LIN {X 0,Y 235.007,Z 550.304,A -85,B 0,C 180,E1 -20010.011,E2 -20010.011} C_VEL
LIN {X 0,Y 236.518,Z 558.697,A -85,B 0,C 180,E1 -20011.333,E2 -20011.333} C_VEL
LIN {X 0,Y 237.232,Z 567.162,A -85,B 0,C 180,E1 -20012.793,E2 -20012.793} C_VEL
LIN {X 0,Y 237.343,Z 573.309,A -85,B 0,C 180,E1 -20013.991,E2 -20013.991} C_VEL
LIN {X 0,Y 235.455,Z 581.31,A -85,B 0,C 180,E1 -20015.572,E2 -20015.572} C_VEL
LIN {X 0,Y 233.143,Z 590.008,A -85,B 0,C 180,E1 -20017.763,E2 -20017.763} C_VEL
LIN {X 0,Y 231.134,Z 596.788,A -85,B 0,C 180,E1 -20020.021,E2 -20020.021} C_VEL
LIN {X 0,Y 230.008,Z 600.386,A -85,B 0,C 180,E1 -20021.472,E2 -20021.472} C_VEL
LIN {X 0,Y 228.59,Z 604.847,A -85,B 0,C 180,E1 -20023.737,E2 -20023.737} C_VEL
LIN {X 0,Y 227.388,Z 608.392,A -85,B 0,C 180,E1 -20026.131,E2 -20026.131} C_VEL
LIN {X 0,Y 226.673,Z 610.489,A -85,B 0,C 180,E1 -20028.084,E2 -20028.084} C_VEL
LIN {X 0,Y 226.284,Z 611.528,A -85,B 0,C 180,E1 -20029.289,E2 -20029.289} C_VEL
LIN {X 0,Y 225.779,Z 612.678,A -85,B 0,C 180,E1 -20031.496,E2 -20031.496} C_VEL
LIN {X 0,Y 225.391,Z 613.018,A -85,B 0,C 180,E1 -20034.166,E2 -20034.166} C_VEL
LIN {X 0,Y 225.298,Z 612.689,A -85,B 0,C 180,E1 -20035.84,E2 -20035.84} C_VEL
LIN {X 0,Y 225.374,Z 611.591,A -85,B 0,C 180,E1 -20037.985,E2 -20037.985} C_VEL
LIN {X 0,Y 225.744,Z 609.19,A -85,B 0,C 180,E1 -20040.659,E2 -20040.659} C_VEL
LIN {X 0,Y 226.275,Z 605.609,A -85,B 0,C 180,E1 -20043.233,E2 -20043.233} C_VEL
LIN {X 0,Y 226.922,Z 600.806,A -85,B 0,C 180,E1 -20045.771,E2 -20045.771} C_VEL
LIN {X 0,Y 227.707,Z 595.856,A -85,B 0,C 180,E1 -20047.809,E2 -20047.809} C_VEL
LIN {X 0,Y 228.959,Z 588.315,A -85,B 0,C 180,E1 -20050.265,E2 -20050.265} C_VEL
LIN {X 0,Y 230.164,Z 580.492,A -85,B 0,C 180,E1 -20052.22,E2 -20052.22} C_VEL
LIN {X 0,Y 231.31,Z 573.319,A -85,B 0,C 180,E1 -20053.676,E2 -20053.676} C_VEL
LIN {X 0,Y 232.129,Z 566.346,A -85,B 0,C 180,E1 -20054.862,E2 -20054.862} C_VEL
LIN {X 0,Y 231.344,Z 557.78,A -85,B 0,C 180,E1 -20056.158,E2 -20056.158} C_VEL
LIN {X 0,Y 230.265,Z 549.339,A -85,B 0,C 180,E1 -20057.215,E2 -20057.215} C_VEL
LIN {X 0,Y 228.715,Z 539.614,A -85,B 0,C 180,E1 -20058.197,E2 -20058.197} C_VEL
LIN {X 0,Y 227.156,Z 531.405,A -85,B 0,C 180,E1 -20058.85,E2 -20058.85} C_VEL
LIN {X 0,Y 227.603,Z 525.746,A -85,B 0,C 180,E1 -20062.904,E2 -20062.904} C_VEL
LIN {X 0,Y 227.945,Z 520.793,A -85,B 0,C 180,E1 -20066.464,E2 -20066.464} C_VEL
LIN {X 0,Y 228.369,Z 516.852,A -85,B 0,C 180,E1 -20069.338,E2 -20069.338} C_VEL
LIN {X 0,Y 228.557,Z 516.827,A -85,B 0,C 180,E1 -20071.761,E2 -20071.761} C_VEL
LIN {X 0,Y 228.36,Z 516.851,A -85,B 0,C 180,E1 -20077.07,E2 -20077.07} C_VEL
LIN {X 0,Y 228.173,Z 516.875,A -85,B 0,C 180,E1 -20080.649,E2 -20080.649} C_VEL
LIN {X 0,Y 228.059,Z 516.89,A -85,B 0,C 180,E1 -20086.101,E2 -20086.101} C_VEL
LIN {X 0,Y 227.943,Z 516.901,A -85,B 0,C 180,E1 -20089.824,E2 -20089.824} C_VEL
LIN {X 0,Y 227.914,Z 516.904,A -85,B 0,C 180,E1 -20093.632,E2 -20093.632} C_VEL
LIN {X 0,Y 227.887,Z 516.909,A -85,B 0,C 180,E1 -20097.554,E2 -20097.554} C_VEL
LIN {X 0,Y 227.873,Z 516.912,A -85,B 0,C 180,E1 -20101.621,E2 -20101.621} C_VEL
LIN {X 0,Y 227.899,Z 516.907,A -85,B 0,C 180,E1 -20105.867,E2 -20105.867} C_VEL
LIN {X 0,Y 227.866,Z 516.912,A -85,B 0,C 180,E1 -20110.367,E2 -20110.367} C_VEL
LIN {X 0,Y 227.899,Z 516.903,A -85,B 0,C 180,E1 -20112.721,E2 -20112.721} C_VEL
LIN {X 0,Y 227.908,Z 516.908,A -85,B 0,C 180,E1 -20117.737,E2 -20117.737} C_VEL
LIN {X 0,Y 227.87,Z 516.91,A -85,B 0,C 180,E1 -20121.914,E2 -20121.914} C_VEL
LIN {X 0,Y 227.889,Z 516.909,A -85,B 0,C 180,E1 -20126.372,E2 -20126.372} C_VEL
LIN {X 0,Y 227.902,Z 516.907,A -85,B 0,C 180,E1 -20130.435,E2 -20130.435} C_VEL
LIN {X 0,Y 227.926,Z 516.904,A -85,B 0,C 180,E1 -20134.425,E2 -20134.425} C_VEL
LIN {X 0,Y 227.96,Z 516.901,A -85,B 0,C 180,E1 -20138.287,E2 -20138.287} C_VEL
LIN {X 0,Y 228.032,Z 516.89,A -85,B 0,C 180,E1 -20142.825,E2 -20142.825} C_VEL
LIN {X 0,Y 228.092,Z 516.885,A -85,B 0,C 180,E1 -20147.544,E2 -20147.544} C_VEL
LIN {X 0,Y 228.323,Z 516.854,A -85,B 0,C 180,E1 -20151.147,E2 -20151.147} C_VEL
LIN {X 0,Y 228.356,Z 516.85,A -85,B 0,C 180,E1 -20152.928,E2 -20152.928} C_VEL
LIN {X 0,Y 228.553,Z 516.82,A -85,B 0,C 180,E1 -20158.238,E2 -20158.238} C_VEL
LIN {X 0,Y 228.553,Z 516.827,A -85,B 0,C 180,E1 -20161.762,E2 -20161.762} C_VEL
LIN {X 0,Y 228.356,Z 516.85,A -85,B 0,C 180,E1 -20167.071,E2 -20167.071} C_VEL
LIN {X 0,Y 228.169,Z 516.874,A -85,B 0,C 180,E1 -20170.65,E2 -20170.65} C_VEL
LIN {X 0,Y 228.055,Z 516.889,A -85,B 0,C 180,E1 -20176.102,E2 -20176.102} C_VEL
LIN {X 0,Y 227.94,Z 516.906,A -85,B 0,C 180,E1 -20179.825,E2 -20179.825} C_VEL
LIN {X 0,Y 227.912,Z 516.911,A -85,B 0,C 180,E1 -20183.633,E2 -20183.633} C_VEL
LIN {X 0,Y 227.883,Z 516.914,A -85,B 0,C 180,E1 -20187.555,E2 -20187.555} C_VEL
LIN {X 0,Y 227.87,Z 516.915,A -85,B 0,C 180,E1 -20191.622,E2 -20191.622} C_VEL
LIN {X 0,Y 227.898,Z 516.909,A -85,B 0,C 180,E1 -20195.869,E2 -20195.869} C_VEL
LIN {X 0,Y 227.835,Z 516.916,A -85,B 0,C 180,E1 -20200.374,E2 -20200.374} C_VEL
LIN {X 0,Y 227.846,Z 516.915,A -85,B 0,C 180,E1 -20204.812,E2 -20204.812} C_VEL
LIN {X 0,Y 227.905,Z 516.909,A -85,B 0,C 180,E1 -20207.74,E2 -20207.74} C_VEL
LIN {X 0,Y 228.276,Z 516.988,A -85,B 0,C 180,E1 -20213.175,E2 -20213.175} C_VEL
LIN {X 0,Y 228.987,Z 520.827,A -85,B 0,C 180,E1 -20216.466,E2 -20216.466} C_VEL
LIN {X 0,Y 228.999,Z 523.333,A -85,B 0,C 180,E1 -20218.553,E2 -20218.553} C_VEL
LIN {X 0,Y 228.777,Z 524.324,A -85,B 0,C 180,E1 -20219.365,E2 -20219.365} C_VEL
LIN {X 0,Y 227.83,Z 525.477,A -85,B 0,C 180,E1 -20220.287,E2 -20220.287} C_VEL
LIN {X 0,Y 224.604,Z 527.281,A -85,B 0,C 180,E1 -20221.709,E2 -20221.709} C_VEL
LIN {X 0,Y 221.378,Z 529.082,A -85,B 0,C 180,E1 -20223.169,E2 -20223.169} C_VEL
LIN {X 0,Y 220.469,Z 530.23,A -85,B 0,C 180,E1 -20224.136,E2 -20224.136} C_VEL
LIN {X 0,Y 220.27,Z 531.464,A -85,B 0,C 180,E1 -20225.118,E2 -20225.118} C_VEL
LIN {X 0,Y 220.333,Z 537.076,A -85,B 0,C 180,E1 -20226.608,E2 -20226.608} C_VEL
LIN {X 0,Y 222.079,Z 549.396,A -85,B 0,C 180,E1 -20227.381,E2 -20227.381} C_VEL
LIN {X 0,Y 223.02,Z 560.406,A -85,B 0,C 180,E1 -20228.39,E2 -20228.39} C_VEL
LIN {X 0,Y 223.44,Z 568.042,A -85,B 0,C 180,E1 -20229.278,E2 -20229.278} C_VEL
LIN {X 0,Y 223.685,Z 576.512,A -85,B 0,C 180,E1 -20230.488,E2 -20230.488} C_VEL
LIN {X 0,Y 223.645,Z 584.746,A -85,B 0,C 180,E1 -20231.923,E2 -20231.923} C_VEL
LIN {X 0,Y 222.623,Z 592.352,A -85,B 0,C 180,E1 -20233.495,E2 -20233.495} C_VEL
LIN {X 0,Y 221.149,Z 601.055,A -85,B 0,C 180,E1 -20235.743,E2 -20235.743} C_VEL
LIN {X 0,Y 220.121,Z 607.776,A -85,B 0,C 180,E1 -20238.023,E2 -20238.023} C_VEL
LIN {X 0,Y 219.513,Z 612.188,A -85,B 0,C 180,E1 -20239.859,E2 -20239.859} C_VEL
LIN {X 0,Y 218.864,Z 617.345,A -85,B 0,C 180,E1 -20242.621,E2 -20242.621} C_VEL
LIN {X 0,Y 218.62,Z 620.919,A -85,B 0,C 180,E1 -20245.244,E2 -20245.244} C_VEL
LIN {X 0,Y 218.634,Z 623.486,A -85,B 0,C 180,E1 -20248.159,E2 -20248.159} C_VEL
LIN {X 0,Y 218.702,Z 624.416,A -85,B 0,C 180,E1 -20250.001,E2 -20250.001} C_VEL
LIN {X 0,Y 218.615,Z 624.76,A -85,B 0,C 180,E1 -20251.843,E2 -20251.843} C_VEL
LIN {X 0,Y 218.602,Z 624.411,A -85,B 0,C 180,E1 -20254.7,E2 -20254.7} C_VEL
LIN {X 0,Y 218.958,Z 622.919,A -85,B 0,C 180,E1 -20257.377,E2 -20257.377} C_VEL
LIN {X 0,Y 219.731,Z 620.18,A -85,B 0,C 180,E1 -20260.133,E2 -20260.133} C_VEL
LIN {X 0,Y 220.4,Z 618.341,A -85,B 0,C 180,E1 -20261.73,E2 -20261.73} C_VEL
LIN {X 0,Y 222.182,Z 617.099,A -85,B 0,C 180,E1 -20264.659,E2 -20264.659} C_VEL
LIN {X 0,Y 223.649,Z 615.845,A -85,B 0,C 180,E1 -20266.429,E2 -20266.429} C_VEL
LIN {X 0,Y 226.461,Z 613.008,A -85,B 0,C 180,E1 -20269.018,E2 -20269.018} C_VEL
LIN {X 0,Y 229.725,Z 609.186,A -85,B 0,C 180,E1 -20271.539,E2 -20271.539} C_VEL
LIN {X 0,Y 233.742,Z 604.208,A -85,B 0,C 180,E1 -20273.949,E2 -20273.949} C_VEL
LIN {X 0,Y 237.155,Z 599.229,A -85,B 0,C 180,E1 -20275.921,E2 -20275.921} C_VEL
LIN {X 0,Y 239.277,Z 594.816,A -85,B 0,C 180,E1 -20277.612,E2 -20277.612} C_VEL
LIN {X 0,Y 241.061,Z 589.316,A -85,B 0,C 180,E1 -20279.712,E2 -20279.712} C_VEL
LIN {X 0,Y 242.574,Z 582.026,A -85,B 0,C 180,E1 -20282.561,E2 -20282.561} C_VEL
LIN {X 0,Y 243.403,Z 575.694,A -85,B 0,C 180,E1 -20285.274,E2 -20285.274} C_VEL
LIN {X 0,Y 243.536,Z 571.75,A -85,B 0,C 180,E1 -20287.303,E2 -20287.303} C_VEL
LIN {X 0,Y 243.563,Z 569.325,A -85,B 0,C 180,E1 -20288.823,E2 -20288.823} C_VEL
LIN {X 0,Y 242.945,Z 566.439,A -85,B 0,C 180,E1 -20291.71,E2 -20291.71} C_VEL
LIN {X 0,Y 242.763,Z 564.841,A -85,B 0,C 180,E1 -20294.012,E2 -20294.012} C_VEL
LIN {X 0,Y 242.779,Z 564.068,A -85,B 0,C 180,E1 -20296.362,E2 -20296.362} C_VEL
LIN {X 0,Y 243.003,Z 564.183,A -85,B 0,C 180,E1 -20298.761,E2 -20298.761} C_VEL
LIN {X 0,Y 243.593,Z 564.891,A -85,B 0,C 180,E1 -20301.169,E2 -20301.169} C_VEL
LIN {X 0,Y 244.177,Z 566.698,A -85,B 0,C 180,E1 -20303.699,E2 -20303.699} C_VEL
LIN {X 0,Y 244.798,Z 569.755,A -85,B 0,C 180,E1 -20306.365,E2 -20306.365} C_VEL
LIN {X 0,Y 245.01,Z 573.587,A -85,B 0,C 180,E1 -20308.914,E2 -20308.914} C_VEL
LIN {X 0,Y 244.673,Z 578.644,A -85,B 0,C 180,E1 -20311.709,E2 -20311.709} C_VEL
LIN {X 0,Y 244.036,Z 582.042,A -85,B 0,C 180,E1 -20313.454,E2 -20313.454} C_VEL
LIN {X 0,Y 239.292,Z 588.328,A -85,B 0,C 180,E1 -20315.721,E2 -20315.721} C_VEL
LIN {X 0,Y 234.2,Z 594.021,A -85,B 0,C 180,E1 -20318.478,E2 -20318.478} C_VEL
LIN {X 0,Y 231.129,Z 596.969,A -85,B 0,C 180,E1 -20320.459,E2 -20320.459} C_VEL
LIN {X 0,Y 228.841,Z 598.849,A -85,B 0,C 180,E1 -20322.115,E2 -20322.115} C_VEL
LIN {X 0,Y 226.793,Z 600.198,A -85,B 0,C 180,E1 -20323.806,E2 -20323.806} C_VEL
LIN {X 0,Y 224.618,Z 601.283,A -85,B 0,C 180,E1 -20325.921,E2 -20325.921} C_VEL
LIN {X 0,Y 221.953,Z 601.744,A -85,B 0,C 180,E1 -20329.048,E2 -20329.048} C_VEL
LIN {X 0,Y 220.221,Z 600.422,A -85,B 0,C 180,E1 -20332.666,E2 -20332.666} C_VEL
LIN {X 0,Y 219.669,Z 599.166,A -85,B 0,C 180,E1 -20334.492,E2 -20334.492} C_VEL
LIN {X 0,Y 219.074,Z 596.298,A -85,B 0,C 180,E1 -20337.242,E2 -20337.242} C_VEL
LIN {X 0,Y 218.812,Z 592.259,A -85,B 0,C 180,E1 -20340,E2 -20340} C_VEL
LIN {X 0,Y 218.961,Z 586.005,A -85,B 0,C 180,E1 -20343.22,E2 -20343.22} C_VEL
LIN {X 0,Y 219.2,Z 578.539,A -85,B 0,C 180,E1 -20346.074,E2 -20346.074} C_VEL
LIN {X 0,Y 219.613,Z 573.028,A -85,B 0,C 180,E1 -20347.817,E2 -20347.817} C_VEL
LIN {X 0,Y 220.038,Z 566.078,A -85,B 0,C 180,E1 -20349.653,E2 -20349.653} C_VEL
LIN {X 0,Y 220.621,Z 557.797,A -85,B 0,C 180,E1 -20351.484,E2 -20351.484} C_VEL
LIN {X 0,Y 221.397,Z 547.795,A -85,B 0,C 180,E1 -20353.306,E2 -20353.306} C_VEL
LIN {X 0,Y 221.702,Z 541.591,A -85,B 0,C 180,E1 -20354.222,E2 -20354.222} C_VEL
LIN {X 0,Y 219.974,Z 529.154,A -85,B 0,C 180,E1 -20355.715,E2 -20355.715} C_VEL
LIN {X 0,Y 219.136,Z 520.974,A -85,B 0,C 180,E1 -20356.487,E2 -20356.487} C_VEL
LIN {X 0,Y 220.969,Z 526.389,A -85,B 0,C 180,E1 -20361.455,E2 -20361.455} C_VEL
LIN {X 0,Y 222.574,Z 531.349,A -85,B 0,C 180,E1 -20365.733,E2 -20365.733} C_VEL
LIN {X 0,Y 222.742,Z 532.104,A -85,B 0,C 180,E1 -20366.214,E2 -20366.214} C_VEL
LIN {X 0,Y 226.254,Z 542.033,A -85,B 0,C 180,E1 -20367.659,E2 -20367.659} C_VEL
LIN {X 0,Y 228.533,Z 550.551,A -85,B 0,C 180,E1 -20368.97,E2 -20368.97} C_VEL
LIN {X 0,Y 230.143,Z 559.812,A -85,B 0,C 180,E1 -20370.51,E2 -20370.51} C_VEL
LIN {X 0,Y 230.849,Z 569.923,A -85,B 0,C 180,E1 -20372.374,E2 -20372.374} C_VEL
LIN {X 0,Y 230.898,Z 573.885,A -85,B 0,C 180,E1 -20373.222,E2 -20373.222} C_VEL
LIN {X 0,Y 229.157,Z 581.225,A -85,B 0,C 180,E1 -20374.72,E2 -20374.72} C_VEL
LIN {X 0,Y 226.671,Z 590.189,A -85,B 0,C 180,E1 -20377.023,E2 -20377.023} C_VEL
LIN {X 0,Y 224.586,Z 596.728,A -85,B 0,C 180,E1 -20379.238,E2 -20379.238} C_VEL
LIN {X 0,Y 223.252,Z 600.783,A -85,B 0,C 180,E1 -20380.928,E2 -20380.928} C_VEL
LIN {X 0,Y 221.759,Z 605.113,A -85,B 0,C 180,E1 -20383.203,E2 -20383.203} C_VEL
LIN {X 0,Y 220.552,Z 608.416,A -85,B 0,C 180,E1 -20385.488,E2 -20385.488} C_VEL
LIN {X 0,Y 219.672,Z 610.803,A -85,B 0,C 180,E1 -20387.788,E2 -20387.788} C_VEL
LIN {X 0,Y 218.878,Z 612.51,A -85,B 0,C 180,E1 -20390.41,E2 -20390.41} C_VEL
LIN {X 0,Y 218.36,Z 613.256,A -85,B 0,C 180,E1 -20393.575,E2 -20393.575} C_VEL
LIN {X 0,Y 218.218,Z 612.326,A -85,B 0,C 180,E1 -20396.863,E2 -20396.863} C_VEL
LIN {X 0,Y 218.572,Z 609.799,A -85,B 0,C 180,E1 -20400.246,E2 -20400.246} C_VEL
LIN {X 0,Y 218.982,Z 607.346,A -85,B 0,C 180,E1 -20402.265,E2 -20402.265} C_VEL
LIN {X 0,Y 219.497,Z 603.602,A -85,B 0,C 180,E1 -20404.625,E2 -20404.625} C_VEL
LIN {X 0,Y 220.285,Z 598.642,A -85,B 0,C 180,E1 -20406.993,E2 -20406.993} C_VEL
LIN {X 0,Y 221.147,Z 593.197,A -85,B 0,C 180,E1 -20409.051,E2 -20409.051} C_VEL
LIN {X 0,Y 222.272,Z 586.681,A -85,B 0,C 180,E1 -20411.04,E2 -20411.04} C_VEL
LIN {X 0,Y 223.435,Z 579.391,A -85,B 0,C 180,E1 -20412.848,E2 -20412.848} C_VEL
LIN {X 0,Y 224.601,Z 571.995,A -85,B 0,C 180,E1 -20414.342,E2 -20414.342} C_VEL
LIN {X 0,Y 225.161,Z 565.964,A -85,B 0,C 180,E1 -20415.378,E2 -20415.378} C_VEL
LIN {X 0,Y 224.376,Z 557.841,A -85,B 0,C 180,E1 -20416.643,E2 -20416.643} C_VEL
LIN {X 0,Y 223.124,Z 548.126,A -85,B 0,C 180,E1 -20417.885,E2 -20417.885} C_VEL
LIN {X 0,Y 221.086,Z 536.223,A -85,B 0,C 180,E1 -20419.062,E2 -20419.062} C_VEL
LIN {X 0,Y 220.183,Z 531.534,A -85,B 0,C 180,E1 -20419.423,E2 -20419.423} C_VEL
LIN {X 0,Y 220.754,Z 524.572,A -85,B 0,C 180,E1 -20424.518,E2 -20424.518} C_VEL
LIN {X 0,Y 221.365,Z 517.725,A -85,B 0,C 180,E1 -20429.544,E2 -20429.544} C_VEL
LIN {X 0,Y 221.515,Z 517.704,A -85,B 0,C 180,E1 -20431.817,E2 -20431.817} C_VEL
LIN {X 0,Y 221.313,Z 517.729,A -85,B 0,C 180,E1 -20437.297,E2 -20437.297} C_VEL
LIN {X 0,Y 221.118,Z 517.753,A -85,B 0,C 180,E1 -20440.993,E2 -20440.993} C_VEL
LIN {X 0,Y 221.017,Z 517.766,A -85,B 0,C 180,E1 -20446.629,E2 -20446.629} C_VEL
LIN {X 0,Y 220.893,Z 517.782,A -85,B 0,C 180,E1 -20450.485,E2 -20450.485} C_VEL
LIN {X 0,Y 220.868,Z 517.785,A -85,B 0,C 180,E1 -20454.434,E2 -20454.434} C_VEL
LIN {X 0,Y 220.838,Z 517.789,A -85,B 0,C 180,E1 -20458.512,E2 -20458.512} C_VEL
LIN {X 0,Y 220.824,Z 517.788,A -85,B 0,C 180,E1 -20462.754,E2 -20462.754} C_VEL
LIN {X 0,Y 220.837,Z 517.787,A -85,B 0,C 180,E1 -20467.287,E2 -20467.287} C_VEL
LIN {X 0,Y 220.839,Z 517.786,A -85,B 0,C 180,E1 -20471.935,E2 -20471.935} C_VEL
LIN {X 0,Y 220.867,Z 517.783,A -85,B 0,C 180,E1 -20477.041,E2 -20477.041} C_VEL
LIN {X 0,Y 220.854,Z 517.784,A -85,B 0,C 180,E1 -20480.473,E2 -20480.473} C_VEL
LIN {X 0,Y 220.814,Z 517.787,A -85,B 0,C 180,E1 -20485.047,E2 -20485.047} C_VEL
LIN {X 0,Y 220.832,Z 517.789,A -85,B 0,C 180,E1 -20489.389,E2 -20489.389} C_VEL
LIN {X 0,Y 220.892,Z 517.779,A -85,B 0,C 180,E1 -20493.549,E2 -20493.549} C_VEL
LIN {X 0,Y 220.876,Z 517.784,A -85,B 0,C 180,E1 -20497.553,E2 -20497.553} C_VEL
LIN {X 0,Y 220.982,Z 517.769,A -85,B 0,C 180,E1 -20502.571,E2 -20502.571} C_VEL
LIN {X 0,Y 221.024,Z 517.763,A -85,B 0,C 180,E1 -20507.139,E2 -20507.139} C_VEL
LIN {X 0,Y 221.255,Z 517.734,A -85,B 0,C 180,E1 -20510.861,E2 -20510.861} C_VEL
LIN {X 0,Y 221.309,Z 517.728,A -85,B 0,C 180,E1 -20512.702,E2 -20512.702} C_VEL
LIN {X 0,Y 221.511,Z 517.697,A -85,B 0,C 180,E1 -20518.182,E2 -20518.182} C_VEL
LIN {X 0,Y 221.511,Z 517.705,A -85,B 0,C 180,E1 -20521.818,E2 -20521.818} C_VEL
LIN {X 0,Y 221.309,Z 517.728,A -85,B 0,C 180,E1 -20527.298,E2 -20527.298} C_VEL
LIN {X 0,Y 221.114,Z 517.753,A -85,B 0,C 180,E1 -20530.994,E2 -20530.994} C_VEL
LIN {X 0,Y 221.014,Z 517.765,A -85,B 0,C 180,E1 -20536.63,E2 -20536.63} C_VEL
LIN {X 0,Y 220.891,Z 517.781,A -85,B 0,C 180,E1 -20540.486,E2 -20540.486} C_VEL
LIN {X 0,Y 220.865,Z 517.785,A -85,B 0,C 180,E1 -20544.435,E2 -20544.435} C_VEL
LIN {X 0,Y 220.833,Z 517.788,A -85,B 0,C 180,E1 -20548.514,E2 -20548.514} C_VEL
LIN {X 0,Y 220.822,Z 517.79,A -85,B 0,C 180,E1 -20552.755,E2 -20552.755} C_VEL
LIN {X 0,Y 220.836,Z 517.789,A -85,B 0,C 180,E1 -20557.288,E2 -20557.288} C_VEL
LIN {X 0,Y 220.811,Z 517.793,A -85,B 0,C 180,E1 -20561.943,E2 -20561.943} C_VEL
LIN {X 0,Y 220.861,Z 517.786,A -85,B 0,C 180,E1 -20567.044,E2 -20567.044} C_VEL
LIN {X 0,Y 221.239,Z 517.741,A -85,B 0,C 180,E1 -20573.338,E2 -20573.338} C_VEL
LIN {X 0,Y 222.053,Z 522.385,A -85,B 0,C 180,E1 -20577.45,E2 -20577.45} C_VEL
LIN {X 0,Y 221.364,Z 525.983,A -85,B 0,C 180,E1 -20580.522,E2 -20580.522} C_VEL
LIN {X 0,Y 220.469,Z 530.23,A -85,B 0,C 180,E1 -20584.136,E2 -20584.136} C_VEL
LIN {X 0,Y 220.051,Z 532.044,A -85,B 0,C 180,E1 -20584.975,E2 -20584.975} C_VEL
LIN {X 0,Y 219.387,Z 534.815,A -85,B 0,C 180,E1 -20585.624,E2 -20585.624} C_VEL
LIN {X 0,Y 218.186,Z 539.974,A -85,B 0,C 180,E1 -20586.306,E2 -20586.306} C_VEL
LIN {X 0,Y 216.312,Z 550.343,A -85,B 0,C 180,E1 -20586.992,E2 -20586.992} C_VEL
LIN {X 0,Y 215.891,Z 556.42,A -85,B 0,C 180,E1 -20587.446,E2 -20587.446} C_VEL
LIN {X 0,Y 215.964,Z 558.354,A -85,B 0,C 180,E1 -20587.645,E2 -20587.645} C_VEL
LIN {X 0,Y 216.515,Z 568.513,A -85,B 0,C 180,E1 -20588.862,E2 -20588.862} C_VEL
LIN {X 0,Y 216.742,Z 576.836,A -85,B 0,C 180,E1 -20590.109,E2 -20590.109} C_VEL
LIN {X 0,Y 216.661,Z 584.849,A -85,B 0,C 180,E1 -20591.564,E2 -20591.564} C_VEL
LIN {X 0,Y 215.894,Z 590.386,A -85,B 0,C 180,E1 -20592.721,E2 -20592.721} C_VEL
LIN {X 0,Y 214.806,Z 596.941,A -85,B 0,C 180,E1 -20594.341,E2 -20594.341} C_VEL
LIN {X 0,Y 213.797,Z 603.161,A -85,B 0,C 180,E1 -20596.213,E2 -20596.213} C_VEL
LIN {X 0,Y 212.955,Z 608.311,A -85,B 0,C 180,E1 -20598.098,E2 -20598.098} C_VEL
LIN {X 0,Y 212.222,Z 613.542,A -85,B 0,C 180,E1 -20600.47,E2 -20600.47} C_VEL
LIN {X 0,Y 211.674,Z 618.363,A -85,B 0,C 180,E1 -20603.328,E2 -20603.328} C_VEL
LIN {X 0,Y 211.493,Z 621.645,A -85,B 0,C 180,E1 -20606.19,E2 -20606.19} C_VEL
LIN {X 0,Y 211.532,Z 623.194,A -85,B 0,C 180,E1 -20608.097,E2 -20608.097} C_VEL
LIN {X 0,Y 211.616,Z 624.139,A -85,B 0,C 180,E1 -20610.001,E2 -20610.001} C_VEL
LIN {X 0,Y 211.513,Z 624.536,A -85,B 0,C 180,E1 -20611.905,E2 -20611.905} C_VEL
LIN {X 0,Y 211.506,Z 624.318,A -85,B 0,C 180,E1 -20614.55,E2 -20614.55} C_VEL
LIN {X 0,Y 211.9,Z 622.876,A -85,B 0,C 180,E1 -20617.625,E2 -20617.625} C_VEL
LIN {X 0,Y 212.724,Z 620.226,A -85,B 0,C 180,E1 -20620.47,E2 -20620.47} C_VEL
LIN {X 0,Y 213.536,Z 617.991,A -85,B 0,C 180,E1 -20622.354,E2 -20622.354} C_VEL
LIN {X 0,Y 215.323,Z 617.118,A -85,B 0,C 180,E1 -20625.137,E2 -20625.137} C_VEL
LIN {X 0,Y 216.845,Z 615.964,A -85,B 0,C 180,E1 -20626.96,E2 -20626.96} C_VEL
LIN {X 0,Y 220.85,Z 612.482,A -85,B 0,C 180,E1 -20630.491,E2 -20630.491} C_VEL
LIN {X 0,Y 224.478,Z 608.648,A -85,B 0,C 180,E1 -20633.04,E2 -20633.04} C_VEL
LIN {X 0,Y 228.891,Z 603.745,A -85,B 0,C 180,E1 -20635.46,E2 -20635.46} C_VEL
LIN {X 0,Y 231.675,Z 599.935,A -85,B 0,C 180,E1 -20637.068,E2 -20637.068} C_VEL
LIN {X 0,Y 234.53,Z 593.822,A -85,B 0,C 180,E1 -20639.655,E2 -20639.655} C_VEL
LIN {X 0,Y 236.494,Z 587.538,A -85,B 0,C 180,E1 -20642.339,E2 -20642.339} C_VEL
LIN {X 0,Y 237.854,Z 581.654,A -85,B 0,C 180,E1 -20644.999,E2 -20644.999} C_VEL
LIN {X 0,Y 238.543,Z 577.23,A -85,B 0,C 180,E1 -20647.3,E2 -20647.3} C_VEL
LIN {X 0,Y 238.777,Z 574.228,A -85,B 0,C 180,E1 -20649.302,E2 -20649.302} C_VEL
LIN {X 0,Y 238.28,Z 571.226,A -85,B 0,C 180,E1 -20652.718,E2 -20652.718} C_VEL
LIN {X 0,Y 238.276,Z 569.993,A -85,B 0,C 180,E1 -20655.064,E2 -20655.064} C_VEL
LIN {X 0,Y 238.369,Z 569.602,A -85,B 0,C 180,E1 -20657.485,E2 -20657.485} C_VEL
LIN {X 0,Y 238.733,Z 569.929,A -85,B 0,C 180,E1 -20659.944,E2 -20659.944} C_VEL
LIN {X 0,Y 239.257,Z 571.123,A -85,B 0,C 180,E1 -20662.478,E2 -20662.478} C_VEL
LIN {X 0,Y 239.574,Z 573.528,A -85,B 0,C 180,E1 -20665.226,E2 -20665.226} C_VEL
LIN {X 0,Y 239.688,Z 575.34,A -85,B 0,C 180,E1 -20666.744,E2 -20666.744} C_VEL
LIN {X 0,Y 239.397,Z 578.979,A -85,B 0,C 180,E1 -20669.28,E2 -20669.28} C_VEL
LIN {X 0,Y 238.505,Z 583.717,A -85,B 0,C 180,E1 -20672.131,E2 -20672.131} C_VEL
LIN {X 0,Y 237.664,Z 585.415,A -85,B 0,C 180,E1 -20672.926,E2 -20672.926} C_VEL
LIN {X 0,Y 233.109,Z 590.652,A -85,B 0,C 180,E1 -20675.034,E2 -20675.034} C_VEL
LIN {X 0,Y 228.574,Z 595.071,A -85,B 0,C 180,E1 -20677.397,E2 -20677.397} C_VEL
LIN {X 0,Y 224.588,Z 598.387,A -85,B 0,C 180,E1 -20679.866,E2 -20679.866} C_VEL
LIN {X 0,Y 222.202,Z 600.031,A -85,B 0,C 180,E1 -20681.562,E2 -20681.562} C_VEL
LIN {X 0,Y 220.082,Z 601.25,A -85,B 0,C 180,E1 -20683.298,E2 -20683.298} C_VEL
LIN {X 0,Y 217.72,Z 602.098,A -85,B 0,C 180,E1 -20685.561,E2 -20685.561} C_VEL
LIN {X 0,Y 215.018,Z 602.075,A -85,B 0,C 180,E1 -20688.69,E2 -20688.69} C_VEL
LIN {X 0,Y 213.942,Z 601.514,A -85,B 0,C 180,E1 -20690.546,E2 -20690.546} C_VEL
LIN {X 0,Y 213.183,Z 600.415,A -85,B 0,C 180,E1 -20692.423,E2 -20692.423} C_VEL
LIN {X 0,Y 212.617,Z 598.906,A -85,B 0,C 180,E1 -20694.309,E2 -20694.309} C_VEL
LIN {X 0,Y 212.015,Z 595.772,A -85,B 0,C 180,E1 -20697.15,E2 -20697.15} C_VEL
LIN {X 0,Y 211.746,Z 591.515,A -85,B 0,C 180,E1 -20700,E2 -20700} C_VEL
LIN {X 0,Y 211.875,Z 585.937,A -85,B 0,C 180,E1 -20702.852,E2 -20702.852} C_VEL
LIN {X 0,Y 212.049,Z 579.653,A -85,B 0,C 180,E1 -20705.342,E2 -20705.342} C_VEL
LIN {X 0,Y 212.553,Z 572.738,A -85,B 0,C 180,E1 -20707.6,E2 -20707.6} C_VEL
LIN {X 0,Y 212.958,Z 565.769,A -85,B 0,C 180,E1 -20709.498,E2 -20709.498} C_VEL
LIN {X 0,Y 213.617,Z 556.39,A -85,B 0,C 180,E1 -20711.626,E2 -20711.626} C_VEL
LIN {X 0,Y 214.421,Z 545.818,A -85,B 0,C 180,E1 -20713.505,E2 -20713.505} C_VEL
LIN {X 0,Y 214.511,Z 541.041,A -85,B 0,C 180,E1 -20714.225,E2 -20714.225} C_VEL
LIN {X 0,Y 212.957,Z 529.999,A -85,B 0,C 180,E1 -20715.583,E2 -20715.583} C_VEL
LIN {X 0,Y 212.2,Z 523.196,A -85,B 0,C 180,E1 -20716.332,E2 -20716.332} C_VEL
LIN {X 0,Y 213.336,Z 526.128,A -85,B 0,C 180,E1 -20719.235,E2 -20719.235} C_VEL
LIN {X 0,Y 215.085,Z 531.076,A -85,B 0,C 180,E1 -20723.805,E2 -20723.805} C_VEL
LIN {X 0,Y 215.495,Z 532.337,A -85,B 0,C 180,E1 -20724.735,E2 -20724.735} C_VEL
LIN {X 0,Y 218.195,Z 537.942,A -85,B 0,C 180,E1 -20725.711,E2 -20725.711} C_VEL
LIN {X 0,Y 221.039,Z 546.782,A -85,B 0,C 180,E1 -20727.149,E2 -20727.149} C_VEL
LIN {X 0,Y 223.131,Z 556.428,A -85,B 0,C 180,E1 -20728.805,E2 -20728.805} C_VEL
LIN {X 0,Y 224.185,Z 564.811,A -85,B 0,C 180,E1 -20730.365,E2 -20730.365} C_VEL
LIN {X 0,Y 224.442,Z 572.456,A -85,B 0,C 180,E1 -20731.93,E2 -20731.93} C_VEL
LIN {X 0,Y 224.38,Z 575.573,A -85,B 0,C 180,E1 -20732.618,E2 -20732.618} C_VEL
LIN {X 0,Y 221.834,Z 585.108,A -85,B 0,C 180,E1 -20734.769,E2 -20734.769} C_VEL
LIN {X 0,Y 219.561,Z 592.256,A -85,B 0,C 180,E1 -20736.846,E2 -20736.846} C_VEL
LIN {X 0,Y 217.455,Z 598.472,A -85,B 0,C 180,E1 -20739.133,E2 -20739.133} C_VEL
LIN {X 0,Y 215.688,Z 603.405,A -85,B 0,C 180,E1 -20741.457,E2 -20741.457} C_VEL
LIN {X 0,Y 214.282,Z 607.226,A -85,B 0,C 180,E1 -20743.816,E2 -20743.816} C_VEL
LIN {X 0,Y 213.013,Z 610.368,A -85,B 0,C 180,E1 -20746.54,E2 -20746.54} C_VEL
LIN {X 0,Y 212.297,Z 611.976,A -85,B 0,C 180,E1 -20748.539,E2 -20748.539} C_VEL
LIN {X 0,Y 211.666,Z 613.098,A -85,B 0,C 180,E1 -20750.885,E2 -20750.885} C_VEL
LIN {X 0,Y 211.296,Z 613.453,A -85,B 0,C 180,E1 -20753.222,E2 -20753.222} C_VEL
LIN {X 0,Y 211.114,Z 612.712,A -85,B 0,C 180,E1 -20756.331,E2 -20756.331} C_VEL
LIN {X 0,Y 211.151,Z 611.943,A -85,B 0,C 180,E1 -20757.821,E2 -20757.821} C_VEL
LIN {X 0,Y 211.437,Z 610.09,A -85,B 0,C 180,E1 -20760.092,E2 -20760.092} C_VEL
LIN {X 0,Y 211.908,Z 607.49,A -85,B 0,C 180,E1 -20762.333,E2 -20762.333} C_VEL
LIN {X 0,Y 212.501,Z 603.201,A -85,B 0,C 180,E1 -20765.058,E2 -20765.058} C_VEL
LIN {X 0,Y 213.285,Z 598.499,A -85,B 0,C 180,E1 -20767.314,E2 -20767.314} C_VEL
LIN {X 0,Y 214.155,Z 593.272,A -85,B 0,C 180,E1 -20769.341,E2 -20769.341} C_VEL
LIN {X 0,Y 215.448,Z 585.941,A -85,B 0,C 180,E1 -20771.613,E2 -20771.613} C_VEL
LIN {X 0,Y 216.702,Z 578.307,A -85,B 0,C 180,E1 -20773.513,E2 -20773.513} C_VEL
LIN {X 0,Y 218.17,Z 568.735,A -85,B 0,C 180,E1 -20775.4,E2 -20775.4} C_VEL
LIN {X 0,Y 217.561,Z 559.482,A -85,B 0,C 180,E1 -20776.93,E2 -20776.93} C_VEL
LIN {X 0,Y 216.559,Z 551.126,A -85,B 0,C 180,E1 -20778.082,E2 -20778.082} C_VEL
LIN {X 0,Y 215.038,Z 541.584,A -85,B 0,C 180,E1 -20779.15,E2 -20779.15} C_VEL
LIN {X 0,Y 213.19,Z 531.641,A -85,B 0,C 180,E1 -20780.033,E2 -20780.033} C_VEL
LIN {X 0,Y 213.826,Z 524.616,A -85,B 0,C 180,E1 -20785.286,E2 -20785.286} C_VEL
LIN {X 0,Y 214.394,Z 518.594,A -85,B 0,C 180,E1 -20789.882,E2 -20789.882} C_VEL
LIN {X 0,Y 214.448,Z 518.585,A -85,B 0,C 180,E1 -20791.877,E2 -20791.877} C_VEL
LIN {X 0,Y 214.25,Z 518.609,A -85,B 0,C 180,E1 -20797.539,E2 -20797.539} C_VEL
LIN {X 0,Y 214.049,Z 518.633,A -85,B 0,C 180,E1 -20801.361,E2 -20801.361} C_VEL
LIN {X 0,Y 213.934,Z 518.647,A -85,B 0,C 180,E1 -20805.236,E2 -20805.236} C_VEL
LIN {X 0,Y 213.84,Z 518.657,A -85,B 0,C 180,E1 -20809.186,E2 -20809.186} C_VEL
LIN {X 0,Y 213.848,Z 518.655,A -85,B 0,C 180,E1 -20813.226,E2 -20813.226} C_VEL
LIN {X 0,Y 213.829,Z 518.66,A -85,B 0,C 180,E1 -20817.449,E2 -20817.449} C_VEL
LIN {X 0,Y 213.779,Z 518.668,A -85,B 0,C 180,E1 -20821.734,E2 -20821.734} C_VEL
LIN {X 0,Y 213.752,Z 518.672,A -85,B 0,C 180,E1 -20826.285,E2 -20826.285} C_VEL
LIN {X 0,Y 213.764,Z 518.666,A -85,B 0,C 180,E1 -20830.871,E2 -20830.871} C_VEL
LIN {X 0,Y 213.807,Z 518.659,A -85,B 0,C 180,E1 -20833.684,E2 -20833.684} C_VEL
LIN {X 0,Y 213.81,Z 518.664,A -85,B 0,C 180,E1 -20836.348,E2 -20836.348} C_VEL
LIN {X 0,Y 213.793,Z 518.664,A -85,B 0,C 180,E1 -20839.118,E2 -20839.118} C_VEL
LIN {X 0,Y 213.753,Z 518.664,A -85,B 0,C 180,E1 -20843.713,E2 -20843.713} C_VEL
LIN {X 0,Y 213.768,Z 518.67,A -85,B 0,C 180,E1 -20848.262,E2 -20848.262} C_VEL
LIN {X 0,Y 213.824,Z 518.658,A -85,B 0,C 180,E1 -20852.603,E2 -20852.603} C_VEL
LIN {X 0,Y 213.85,Z 518.658,A -85,B 0,C 180,E1 -20856.952,E2 -20856.952} C_VEL
LIN {X 0,Y 213.941,Z 518.645,A -85,B 0,C 180,E1 -20862.803,E2 -20862.803} C_VEL
LIN {X 0,Y 213.979,Z 518.641,A -85,B 0,C 180,E1 -20866.708,E2 -20866.708} C_VEL
LIN {X 0,Y 214.194,Z 518.614,A -85,B 0,C 180,E1 -20870.557,E2 -20870.557} C_VEL
LIN {X 0,Y 214.246,Z 518.609,A -85,B 0,C 180,E1 -20872.46,E2 -20872.46} C_VEL
LIN {X 0,Y 214.445,Z 518.578,A -85,B 0,C 180,E1 -20878.122,E2 -20878.122} C_VEL
LIN {X 0,Y 214.548,Z 518.569,A -85,B 0,C 180,E1 -20880,E2 -20880} C_VEL
LIN {X 0,Y 214.445,Z 518.585,A -85,B 0,C 180,E1 -20881.878,E2 -20881.878} C_VEL
LIN {X 0,Y 214.246,Z 518.61,A -85,B 0,C 180,E1 -20887.54,E2 -20887.54} C_VEL
LIN {X 0,Y 214.045,Z 518.635,A -85,B 0,C 180,E1 -20891.362,E2 -20891.362} C_VEL
LIN {X 0,Y 213.931,Z 518.649,A -85,B 0,C 180,E1 -20895.237,E2 -20895.237} C_VEL
LIN {X 0,Y 213.838,Z 518.662,A -85,B 0,C 180,E1 -20899.187,E2 -20899.187} C_VEL
LIN {X 0,Y 213.845,Z 518.661,A -85,B 0,C 180,E1 -20903.227,E2 -20903.227} C_VEL
LIN {X 0,Y 213.826,Z 518.665,A -85,B 0,C 180,E1 -20907.45,E2 -20907.45} C_VEL
LIN {X 0,Y 213.777,Z 518.67,A -85,B 0,C 180,E1 -20911.736,E2 -20911.736} C_VEL
LIN {X 0,Y 213.75,Z 518.67,A -85,B 0,C 180,E1 -20916.287,E2 -20916.287} C_VEL
LIN {X 0,Y 213.736,Z 518.674,A -85,B 0,C 180,E1 -20921.119,E2 -20921.119} C_VEL
LIN {X 0,Y 213.773,Z 518.67,A -85,B 0,C 180,E1 -20923.676,E2 -20923.676} C_VEL
LIN {X 0,Y 213.778,Z 518.668,A -85,B 0,C 180,E1 -20926.341,E2 -20926.341} C_VEL
LIN {X 0,Y 214.043,Z 518.637,A -85,B 0,C 180,E1 -20932.001,E2 -20932.001} C_VEL
LIN {X 0,Y 214.257,Z 518.752,A -85,B 0,C 180,E1 -20933.814,E2 -20933.814} C_VEL
LIN {X 0,Y 214.958,Z 522.63,A -85,B 0,C 180,E1 -20937.355,E2 -20937.355} C_VEL
LIN {X 0,Y 214.252,Z 526.21,A -85,B 0,C 180,E1 -20940.527,E2 -20940.527} C_VEL
LIN {X 0,Y 213.358,Z 530.376,A -85,B 0,C 180,E1 -20944.123,E2 -20944.123} C_VEL
LIN {X 0,Y 213.392,Z 537.001,A -85,B 0,C 180,E1 -20946.012,E2 -20946.012} C_VEL
LIN {X 0,Y 215.18,Z 549.287,A -85,B 0,C 180,E1 -20946.816,E2 -20946.816} C_VEL
LIN {X 0,Y 215.964,Z 558.354,A -85,B 0,C 180,E1 -20947.645,E2 -20947.645} C_VEL
LIN {X 0,Y 215.681,Z 564.161,A -85,B 0,C 180,E1 -20948.241,E2 -20948.241} C_VEL
LIN {X 0,Y 214.375,Z 569.616,A -85,B 0,C 180,E1 -20948.837,E2 -20948.837} C_VEL
LIN {X 0,Y 210.899,Z 579.738,A -85,B 0,C 180,E1 -20950.224,E2 -20950.224} C_VEL
LIN {X 0,Y 209.778,Z 584.404,A -85,B 0,C 180,E1 -20951.083,E2 -20951.083} C_VEL
LIN {X 0,Y 209.641,Z 585.944,A -85,B 0,C 180,E1 -20951.391,E2 -20951.391} C_VEL
LIN {X 0,Y 208.299,Z 594.378,A -85,B 0,C 180,E1 -20953.335,E2 -20953.335} C_VEL
LIN {X 0,Y 206.865,Z 602.404,A -85,B 0,C 180,E1 -20955.742,E2 -20955.742} C_VEL
LIN {X 0,Y 206.004,Z 607.651,A -85,B 0,C 180,E1 -20957.69,E2 -20957.69} C_VEL
LIN {X 0,Y 205.198,Z 612.963,A -85,B 0,C 180,E1 -20960.141,E2 -20960.141} C_VEL
LIN {X 0,Y 204.763,Z 616.368,A -85,B 0,C 180,E1 -20962.11,E2 -20962.11} C_VEL
LIN {X 0,Y 204.516,Z 619.122,A -85,B 0,C 180,E1 -20964.084,E2 -20964.084} C_VEL
LIN {X 0,Y 204.424,Z 621.287,A -85,B 0,C 180,E1 -20966.058,E2 -20966.058} C_VEL
LIN {X 0,Y 204.432,Z 622.868,A -85,B 0,C 180,E1 -20968.031,E2 -20968.031} C_VEL
LIN {X 0,Y 204.531,Z 623.845,A -85,B 0,C 180,E1 -20970.001,E2 -20970.001} C_VEL
LIN {X 0,Y 204.414,Z 624.309,A -85,B 0,C 180,E1 -20971.971,E2 -20971.971} C_VEL
LIN {X 0,Y 204.411,Z 624.217,A -85,B 0,C 180,E1 -20974.388,E2 -20974.388} C_VEL
LIN {X 0,Y 204.574,Z 623.82,A -85,B 0,C 180,E1 -20975.917,E2 -20975.917} C_VEL
LIN {X 0,Y 204.868,Z 622.813,A -85,B 0,C 180,E1 -20977.888,E2 -20977.888} C_VEL
LIN {X 0,Y 205.741,Z 620.273,A -85,B 0,C 180,E1 -20980.83,E2 -20980.83} C_VEL
LIN {X 0,Y 206.885,Z 617.51,A -85,B 0,C 180,E1 -20983.257,E2 -20983.257} C_VEL
LIN {X 0,Y 208.485,Z 616.932,A -85,B 0,C 180,E1 -20985.646,E2 -20985.646} C_VEL
LIN {X 0,Y 212.014,Z 614.769,A -85,B 0,C 180,E1 -20989.36,E2 -20989.36} C_VEL
LIN {X 0,Y 215.467,Z 611.98,A -85,B 0,C 180,E1 -20992.032,E2 -20992.032} C_VEL
LIN {X 0,Y 219.455,Z 608.234,A -85,B 0,C 180,E1 -20994.604,E2 -20994.604} C_VEL
LIN {X 0,Y 222.62,Z 605.157,A -85,B 0,C 180,E1 -20996.231,E2 -20996.231} C_VEL
LIN {X 0,Y 225.548,Z 601.63,A -85,B 0,C 180,E1 -20997.866,E2 -20997.866} C_VEL
LIN {X 0,Y 228.117,Z 597.118,A -85,B 0,C 180,E1 -20999.975,E2 -20999.975} C_VEL
LIN {X 0,Y 230.223,Z 592.185,A -85,B 0,C 180,E1 -21002.292,E2 -21002.292} C_VEL
LIN {X 0,Y 232.18,Z 586.273,A -85,B 0,C 180,E1 -21005.187,E2 -21005.187} C_VEL
LIN {X 0,Y 233.388,Z 581.656,A -85,B 0,C 180,E1 -21007.782,E2 -21007.782} C_VEL
LIN {X 0,Y 233.676,Z 578.66,A -85,B 0,C 180,E1 -21010.014,E2 -21010.014} C_VEL
LIN {X 0,Y 233.469,Z 575.946,A -85,B 0,C 180,E1 -21013.818,E2 -21013.818} C_VEL
LIN {X 0,Y 233.55,Z 575.05,A -85,B 0,C 180,E1 -21016.238,E2 -21016.238} C_VEL
LIN {X 0,Y 233.699,Z 574.96,A -85,B 0,C 180,E1 -21018.75,E2 -21018.75} C_VEL
LIN {X 0,Y 234.051,Z 575.624,A -85,B 0,C 180,E1 -21021.328,E2 -21021.328} C_VEL
LIN {X 0,Y 234.312,Z 577.41,A -85,B 0,C 180,E1 -21024.082,E2 -21024.082} C_VEL
LIN {X 0,Y 234.254,Z 579.683,A -85,B 0,C 180,E1 -21026.403,E2 -21026.403} C_VEL
LIN {X 0,Y 233.593,Z 583.386,A -85,B 0,C 180,E1 -21029.238,E2 -21029.238} C_VEL
LIN {X 0,Y 232.813,Z 586.212,A -85,B 0,C 180,E1 -21031.119,E2 -21031.119} C_VEL
LIN {X 0,Y 232.131,Z 587.507,A -85,B 0,C 180,E1 -21031.911,E2 -21031.911} C_VEL
LIN {X 0,Y 226.927,Z 592.809,A -85,B 0,C 180,E1 -21034.305,E2 -21034.305} C_VEL
LIN {X 0,Y 222.233,Z 596.886,A -85,B 0,C 180,E1 -21036.715,E2 -21036.715} C_VEL
LIN {X 0,Y 218.067,Z 599.836,A -85,B 0,C 180,E1 -21039.236,E2 -21039.236} C_VEL
LIN {X 0,Y 213.363,Z 602.1,A -85,B 0,C 180,E1 -21042.756,E2 -21042.756} C_VEL
LIN {X 0,Y 211.365,Z 602.664,A -85,B 0,C 180,E1 -21044.573,E2 -21044.573} C_VEL
LIN {X 0,Y 209.668,Z 602.72,A -85,B 0,C 180,E1 -21046.43,E2 -21046.43} C_VEL
LIN {X 0,Y 207.749,Z 602.166,A -85,B 0,C 180,E1 -21048.832,E2 -21048.832} C_VEL
LIN {X 0,Y 206.151,Z 600.344,A -85,B 0,C 180,E1 -21052.163,E2 -21052.163} C_VEL
LIN {X 0,Y 205.328,Z 597.638,A -85,B 0,C 180,E1 -21055.091,E2 -21055.091} C_VEL
LIN {X 0,Y 204.816,Z 593.781,A -85,B 0,C 180,E1 -21058.034,E2 -21058.034} C_VEL
LIN {X 0,Y 204.728,Z 588.726,A -85,B 0,C 180,E1 -21060.984,E2 -21060.984} C_VEL
LIN {X 0,Y 204.913,Z 583.474,A -85,B 0,C 180,E1 -21063.441,E2 -21063.441} C_VEL
LIN {X 0,Y 205.11,Z 577.017,A -85,B 0,C 180,E1 -21065.9,E2 -21065.9} C_VEL
LIN {X 0,Y 205.675,Z 569.117,A -85,B 0,C 180,E1 -21068.35,E2 -21068.35} C_VEL
LIN {X 0,Y 206.259,Z 560.253,A -85,B 0,C 180,E1 -21070.553,E2 -21070.553} C_VEL
LIN {X 0,Y 206.89,Z 552.013,A -85,B 0,C 180,E1 -21072.258,E2 -21072.258} C_VEL
LIN {X 0,Y 207.493,Z 543.552,A -85,B 0,C 180,E1 -21073.715,E2 -21073.715} C_VEL
LIN {X 0,Y 206.941,Z 538.083,A -85,B 0,C 180,E1 -21074.505,E2 -21074.505} C_VEL
LIN {X 0,Y 205.555,Z 527.673,A -85,B 0,C 180,E1 -21075.747,E2 -21075.747} C_VEL
LIN {X 0,Y 205.315,Z 525.289,A -85,B 0,C 180,E1 -21076.055,E2 -21076.055} C_VEL
LIN {X 0,Y 206.489,Z 527.988,A -85,B 0,C 180,E1 -21078.865,E2 -21078.865} C_VEL
LIN {X 0,Y 207.993,Z 532.265,A -85,B 0,C 180,E1 -21082.998,E2 -21082.998} C_VEL
LIN {X 0,Y 209.781,Z 535.779,A -85,B 0,C 180,E1 -21083.705,E2 -21083.705} C_VEL
LIN {X 0,Y 211.307,Z 538.304,A -85,B 0,C 180,E1 -21084.257,E2 -21084.257} C_VEL
LIN {X 0,Y 213.553,Z 543.35,A -85,B 0,C 180,E1 -21085.268,E2 -21085.268} C_VEL
LIN {X 0,Y 215.906,Z 552.295,A -85,B 0,C 180,E1 -21086.85,E2 -21086.85} C_VEL
LIN {X 0,Y 217.383,Z 560.965,A -85,B 0,C 180,E1 -21088.481,E2 -21088.481} C_VEL
LIN {X 0,Y 218.1,Z 570.544,A -85,B 0,C 180,E1 -21090.446,E2 -21090.446} C_VEL
LIN {X 0,Y 217.985,Z 576.351,A -85,B 0,C 180,E1 -21091.775,E2 -21091.775} C_VEL
LIN {X 0,Y 215.855,Z 584.318,A -85,B 0,C 180,E1 -21093.608,E2 -21093.608} C_VEL
LIN {X 0,Y 213.385,Z 591.838,A -85,B 0,C 180,E1 -21095.805,E2 -21095.805} C_VEL
LIN {X 0,Y 211.383,Z 597.425,A -85,B 0,C 180,E1 -21097.848,E2 -21097.848} C_VEL
LIN {X 0,Y 209.863,Z 601.403,A -85,B 0,C 180,E1 -21099.624,E2 -21099.624} C_VEL
LIN {X 0,Y 208.158,Z 605.671,A -85,B 0,C 180,E1 -21102.03,E2 -21102.03} C_VEL
LIN {X 0,Y 206.802,Z 608.931,A -85,B 0,C 180,E1 -21104.464,E2 -21104.464} C_VEL
LIN {X 0,Y 205.737,Z 611.277,A -85,B 0,C 180,E1 -21106.904,E2 -21106.904} C_VEL
LIN {X 0,Y 204.974,Z 612.785,A -85,B 0,C 180,E1 -21109.347,E2 -21109.347} C_VEL
LIN {X 0,Y 204.323,Z 613.576,A -85,B 0,C 180,E1 -21112.29,E2 -21112.29} C_VEL
LIN {X 0,Y 204.023,Z 613.091,A -85,B 0,C 180,E1 -21115.765,E2 -21115.765} C_VEL
LIN {X 0,Y 204.218,Z 610.836,A -85,B 0,C 180,E1 -21119.357,E2 -21119.357} C_VEL
LIN {X 0,Y 204.772,Z 607.79,A -85,B 0,C 180,E1 -21122.25,E2 -21122.25} C_VEL
LIN {X 0,Y 205.434,Z 603.275,A -85,B 0,C 180,E1 -21125.223,E2 -21125.223} C_VEL
LIN {X 0,Y 206.233,Z 598.6,A -85,B 0,C 180,E1 -21127.533,E2 -21127.533} C_VEL
LIN {X 0,Y 207.144,Z 593.298,A -85,B 0,C 180,E1 -21129.648,E2 -21129.648} C_VEL
LIN {X 0,Y 208.205,Z 587.549,A -85,B 0,C 180,E1 -21131.532,E2 -21131.532} C_VEL
LIN {X 0,Y 209.388,Z 580.513,A -85,B 0,C 180,E1 -21133.422,E2 -21133.422} C_VEL
LIN {X 0,Y 210.806,Z 572.301,A -85,B 0,C 180,E1 -21135.2,E2 -21135.2} C_VEL
LIN {X 0,Y 211.287,Z 568.635,A -85,B 0,C 180,E1 -21135.898,E2 -21135.898} C_VEL
LIN {X 0,Y 210.621,Z 559.992,A -85,B 0,C 180,E1 -21137.385,E2 -21137.385} C_VEL
LIN {X 0,Y 209.561,Z 551.192,A -85,B 0,C 180,E1 -21138.643,E2 -21138.643} C_VEL
LIN {X 0,Y 208.078,Z 541.721,A -85,B 0,C 180,E1 -21139.741,E2 -21139.741} C_VEL
LIN {X 0,Y 206.221,Z 531.813,A -85,B 0,C 180,E1 -21140.636,E2 -21140.636} C_VEL
LIN {X 0,Y 206.788,Z 525.935,A -85,B 0,C 180,E1 -21145.125,E2 -21145.125} C_VEL
LIN {X 0,Y 207.387,Z 519.468,A -85,B 0,C 180,E1 -21150.242,E2 -21150.242} C_VEL
LIN {X 0,Y 207.385,Z 519.465,A -85,B 0,C 180,E1 -21151.941,E2 -21151.941} C_VEL
LIN {X 0,Y 207.19,Z 519.489,A -85,B 0,C 180,E1 -21157.797,E2 -21157.797} C_VEL
LIN {X 0,Y 206.984,Z 519.514,A -85,B 0,C 180,E1 -21161.754,E2 -21161.754} C_VEL
LIN {X 0,Y 206.868,Z 519.528,A -85,B 0,C 180,E1 -21165.77,E2 -21165.77} C_VEL
LIN {X 0,Y 206.784,Z 519.537,A -85,B 0,C 180,E1 -21169.868,E2 -21169.868} C_VEL
LIN {X 0,Y 206.764,Z 519.54,A -85,B 0,C 180,E1 -21174.071,E2 -21174.071} C_VEL
LIN {X 0,Y 206.744,Z 519.545,A -85,B 0,C 180,E1 -21178.418,E2 -21178.418} C_VEL
LIN {X 0,Y 206.709,Z 519.546,A -85,B 0,C 180,E1 -21182.955,E2 -21182.955} C_VEL
LIN {X 0,Y 206.72,Z 519.547,A -85,B 0,C 180,E1 -21187.73,E2 -21187.73} C_VEL
LIN {X 0,Y 206.705,Z 519.542,A -85,B 0,C 180,E1 -21192.842,E2 -21192.842} C_VEL
LIN {X 0,Y 206.714,Z 519.546,A -85,B 0,C 180,E1 -21197.158,E2 -21197.158} C_VEL
LIN {X 0,Y 206.758,Z 519.539,A -85,B 0,C 180,E1 -21201.424,E2 -21201.424} C_VEL
LIN {X 0,Y 206.729,Z 519.541,A -85,B 0,C 180,E1 -21204.694,E2 -21204.694} C_VEL
LIN {X 0,Y 206.705,Z 519.548,A -85,B 0,C 180,E1 -21209.336,E2 -21209.336} C_VEL
LIN {X 0,Y 206.73,Z 519.543,A -85,B 0,C 180,E1 -21213.772,E2 -21213.772} C_VEL
LIN {X 0,Y 206.756,Z 519.543,A -85,B 0,C 180,E1 -21218.043,E2 -21218.043} C_VEL
LIN {X 0,Y 206.871,Z 519.528,A -85,B 0,C 180,E1 -21222.196,E2 -21222.196} C_VEL
LIN {X 0,Y 206.912,Z 519.522,A -85,B 0,C 180,E1 -21226.245,E2 -21226.245} C_VEL
LIN {X 0,Y 207.13,Z 519.495,A -85,B 0,C 180,E1 -21230.232,E2 -21230.232} C_VEL
LIN {X 0,Y 207.186,Z 519.489,A -85,B 0,C 180,E1 -21232.202,E2 -21232.202} C_VEL
LIN {X 0,Y 207.381,Z 519.457,A -85,B 0,C 180,E1 -21238.058,E2 -21238.058} C_VEL
LIN {X 0,Y 207.513,Z 519.445,A -85,B 0,C 180,E1 -21240,E2 -21240} C_VEL
LIN {X 0,Y 207.381,Z 519.465,A -85,B 0,C 180,E1 -21241.942,E2 -21241.942} C_VEL
LIN {X 0,Y 207.186,Z 519.49,A -85,B 0,C 180,E1 -21247.798,E2 -21247.798} C_VEL
LIN {X 0,Y 206.981,Z 519.516,A -85,B 0,C 180,E1 -21251.755,E2 -21251.755} C_VEL
LIN {X 0,Y 206.865,Z 519.531,A -85,B 0,C 180,E1 -21255.771,E2 -21255.771} C_VEL
LIN {X 0,Y 206.782,Z 519.541,A -85,B 0,C 180,E1 -21259.869,E2 -21259.869} C_VEL
LIN {X 0,Y 206.761,Z 519.543,A -85,B 0,C 180,E1 -21264.072,E2 -21264.072} C_VEL
LIN {X 0,Y 206.741,Z 519.544,A -85,B 0,C 180,E1 -21268.419,E2 -21268.419} C_VEL
LIN {X 0,Y 206.707,Z 519.549,A -85,B 0,C 180,E1 -21272.956,E2 -21272.956} C_VEL
LIN {X 0,Y 206.719,Z 519.548,A -85,B 0,C 180,E1 -21275.321,E2 -21275.321} C_VEL
LIN {X 0,Y 206.675,Z 519.552,A -85,B 0,C 180,E1 -21280.248,E2 -21280.248} C_VEL
LIN {X 0,Y 206.683,Z 519.551,A -85,B 0,C 180,E1 -21284.434,E2 -21284.434} C_VEL
LIN {X 0,Y 206.811,Z 519.537,A -85,B 0,C 180,E1 -21289.785,E2 -21289.785} C_VEL
LIN {X 0,Y 207.248,Z 519.578,A -85,B 0,C 180,E1 -21294.172,E2 -21294.172} C_VEL
LIN {X 0,Y 207.803,Z 523.356,A -85,B 0,C 180,E1 -21297.726,E2 -21297.726} C_VEL
LIN {X 0,Y 206.702,Z 528.157,A -85,B 0,C 180,E1 -21302.131,E2 -21302.131} C_VEL
LIN {X 0,Y 206.512,Z 529.108,A -85,B 0,C 180,E1 -21302.999,E2 -21302.999} C_VEL
LIN {X 0,Y 206.417,Z 536.65,A -85,B 0,C 180,E1 -21305.359,E2 -21305.359} C_VEL
LIN {X 0,Y 208.356,Z 549.647,A -85,B 0,C 180,E1 -21306.279,E2 -21306.279} C_VEL
LIN {X 0,Y 209.129,Z 559.433,A -85,B 0,C 180,E1 -21307.231,E2 -21307.231} C_VEL
LIN {X 0,Y 209.585,Z 568.42,A -85,B 0,C 180,E1 -21308.356,E2 -21308.356} C_VEL
LIN {X 0,Y 209.807,Z 577.09,A -85,B 0,C 180,E1 -21309.706,E2 -21309.706} C_VEL
LIN {X 0,Y 209.641,Z 585.944,A -85,B 0,C 180,E1 -21311.391,E2 -21311.391} C_VEL
LIN {X 0,Y 209.116,Z 589.05,A -85,B 0,C 180,E1 -21312.031,E2 -21312.031} C_VEL
LIN {X 0,Y 207.963,Z 592.003,A -85,B 0,C 180,E1 -21312.672,E2 -21312.672} C_VEL
LIN {X 0,Y 204.619,Z 597.422,A -85,B 0,C 180,E1 -21313.997,E2 -21313.997} C_VEL
LIN {X 0,Y 200.402,Z 603.53,A -85,B 0,C 180,E1 -21315.903,E2 -21315.903} C_VEL
LIN {X 0,Y 199.049,Z 606.953,A -85,B 0,C 180,E1 -21317.248,E2 -21317.248} C_VEL
LIN {X 0,Y 198.194,Z 612.366,A -85,B 0,C 180,E1 -21319.788,E2 -21319.788} C_VEL
LIN {X 0,Y 197.714,Z 615.854,A -85,B 0,C 180,E1 -21321.827,E2 -21321.827} C_VEL
LIN {X 0,Y 197.354,Z 619.942,A -85,B 0,C 180,E1 -21324.996,E2 -21324.996} C_VEL
LIN {X 0,Y 197.336,Z 622.517,A -85,B 0,C 180,E1 -21327.96,E2 -21327.96} C_VEL
LIN {X 0,Y 197.447,Z 623.551,A -85,B 0,C 180,E1 -21330.001,E2 -21330.001} C_VEL
LIN {X 0,Y 197.319,Z 624.081,A -85,B 0,C 180,E1 -21332.042,E2 -21332.042} C_VEL
LIN {X 0,Y 197.311,Z 624.12,A -85,B 0,C 180,E1 -21334.19,E2 -21334.19} C_VEL
LIN {X 0,Y 197.508,Z 623.721,A -85,B 0,C 180,E1 -21336.129,E2 -21336.129} C_VEL
LIN {X 0,Y 197.815,Z 622.731,A -85,B 0,C 180,E1 -21338.171,E2 -21338.171} C_VEL
LIN {X 0,Y 198.777,Z 620.333,A -85,B 0,C 180,E1 -21341.214,E2 -21341.214} C_VEL
LIN {X 0,Y 200.212,Z 616.976,A -85,B 0,C 180,E1 -21344.096,E2 -21344.096} C_VEL
LIN {X 0,Y 203.297,Z 616.077,A -85,B 0,C 180,E1 -21348.128,E2 -21348.128} C_VEL
LIN {X 0,Y 207.642,Z 613.433,A -85,B 0,C 180,E1 -21351.859,E2 -21351.859} C_VEL
LIN {X 0,Y 211.617,Z 610.397,A -85,B 0,C 180,E1 -21354.529,E2 -21354.529} C_VEL
LIN {X 0,Y 217.931,Z 604.893,A -85,B 0,C 180,E1 -21357.88,E2 -21357.88} C_VEL
LIN {X 0,Y 219.447,Z 603.178,A -85,B 0,C 180,E1 -21358.712,E2 -21358.712} C_VEL
LIN {X 0,Y 222.453,Z 598.669,A -85,B 0,C 180,E1 -21361.073,E2 -21361.073} C_VEL
LIN {X 0,Y 225.328,Z 592.808,A -85,B 0,C 180,E1 -21364.155,E2 -21364.155} C_VEL
LIN {X 0,Y 227.369,Z 587.689,A -85,B 0,C 180,E1 -21367.067,E2 -21367.067} C_VEL
LIN {X 0,Y 228.106,Z 585.24,A -85,B 0,C 180,E1 -21368.693,E2 -21368.693} C_VEL
LIN {X 0,Y 228.442,Z 583.385,A -85,B 0,C 180,E1 -21370.246,E2 -21370.246} C_VEL
LIN {X 0,Y 228.344,Z 581.696,A -85,B 0,C 180,E1 -21372.62,E2 -21372.62} C_VEL
LIN {X 0,Y 228.433,Z 580.519,A -85,B 0,C 180,E1 -21375.043,E2 -21375.043} C_VEL
LIN {X 0,Y 228.572,Z 579.993,A -85,B 0,C 180,E1 -21377.557,E2 -21377.557} C_VEL
LIN {X 0,Y 228.751,Z 580.228,A -85,B 0,C 180,E1 -21380.183,E2 -21380.183} C_VEL
LIN {X 0,Y 228.97,Z 581.343,A -85,B 0,C 180,E1 -21382.945,E2 -21382.945} C_VEL
LIN {X 0,Y 228.696,Z 583.86,A -85,B 0,C 180,E1 -21386.072,E2 -21386.072} C_VEL
LIN {X 0,Y 227.481,Z 587.718,A -85,B 0,C 180,E1 -21389.353,E2 -21389.353} C_VEL
LIN {X 0,Y 226.527,Z 589.677,A -85,B 0,C 180,E1 -21390.852,E2 -21390.852} C_VEL
LIN {X 0,Y 224.28,Z 591.979,A -85,B 0,C 180,E1 -21391.963,E2 -21391.963} C_VEL
LIN {X 0,Y 219.117,Z 596.271,A -85,B 0,C 180,E1 -21394.342,E2 -21394.342} C_VEL
LIN {X 0,Y 214.36,Z 599.492,A -85,B 0,C 180,E1 -21396.832,E2 -21396.832} C_VEL
LIN {X 0,Y 208.96,Z 602.288,A -85,B 0,C 180,E1 -21400.347,E2 -21400.347} C_VEL
LIN {X 0,Y 204.574,Z 603.202,A -85,B 0,C 180,E1 -21404.048,E2 -21404.048} C_VEL
LIN {X 0,Y 202.807,Z 603.098,A -85,B 0,C 180,E1 -21405.962,E2 -21405.962} C_VEL
LIN {X 0,Y 200.48,Z 601.999,A -85,B 0,C 180,E1 -21408.986,E2 -21408.986} C_VEL
LIN {X 0,Y 199.127,Z 600.047,A -85,B 0,C 180,E1 -21411.884,E2 -21411.884} C_VEL
LIN {X 0,Y 198.293,Z 597.032,A -85,B 0,C 180,E1 -21414.917,E2 -21414.917} C_VEL
LIN {X 0,Y 197.763,Z 592.939,A -85,B 0,C 180,E1 -21417.964,E2 -21417.964} C_VEL
LIN {X 0,Y 197.714,Z 587.618,A -85,B 0,C 180,E1 -21421.019,E2 -21421.019} C_VEL
LIN {X 0,Y 197.926,Z 580.73,A -85,B 0,C 180,E1 -21424.073,E2 -21424.073} C_VEL
LIN {X 0,Y 198.343,Z 572.88,A -85,B 0,C 180,E1 -21426.842,E2 -21426.842} C_VEL
LIN {X 0,Y 198.838,Z 564.914,A -85,B 0,C 180,E1 -21429.152,E2 -21429.152} C_VEL
LIN {X 0,Y 199.506,Z 555.143,A -85,B 0,C 180,E1 -21431.429,E2 -21431.429} C_VEL
LIN {X 0,Y 200.273,Z 545.731,A -85,B 0,C 180,E1 -21433.185,E2 -21433.185} C_VEL
LIN {X 0,Y 200.307,Z 540.988,A -85,B 0,C 180,E1 -21433.959,E2 -21433.959} C_VEL
LIN {X 0,Y 198.735,Z 529.938,A -85,B 0,C 180,E1 -21435.381,E2 -21435.381} C_VEL
LIN {X 0,Y 198.429,Z 527.388,A -85,B 0,C 180,E1 -21435.668,E2 -21435.668} C_VEL
LIN {X 0,Y 199.644,Z 529.896,A -85,B 0,C 180,E1 -21438.471,E2 -21438.471} C_VEL
LIN {X 0,Y 200.588,Z 532.572,A -85,B 0,C 180,E1 -21441.114,E2 -21441.114} C_VEL
LIN {X 0,Y 202.608,Z 536.256,A -85,B 0,C 180,E1 -21441.961,E2 -21441.961} C_VEL
LIN {X 0,Y 203.949,Z 538.309,A -85,B 0,C 180,E1 -21442.476,E2 -21442.476} C_VEL
LIN {X 0,Y 207.517,Z 545.116,A -85,B 0,C 180,E1 -21444.096,E2 -21444.096} C_VEL
LIN {X 0,Y 209.844,Z 553.926,A -85,B 0,C 180,E1 -21445.81,E2 -21445.81} C_VEL
LIN {X 0,Y 211.355,Z 563.503,A -85,B 0,C 180,E1 -21447.745,E2 -21447.745} C_VEL
LIN {X 0,Y 211.775,Z 572.87,A -85,B 0,C 180,E1 -21449.854,E2 -21449.854} C_VEL
LIN {X 0,Y 211.383,Z 578.873,A -85,B 0,C 180,E1 -21451.311,E2 -21451.311} C_VEL
LIN {X 0,Y 208.99,Z 586.503,A -85,B 0,C 180,E1 -21453.225,E2 -21453.225} C_VEL
LIN {X 0,Y 206.568,Z 593.274,A -85,B 0,C 180,E1 -21455.337,E2 -21455.337} C_VEL
LIN {X 0,Y 204.261,Z 599.225,A -85,B 0,C 180,E1 -21457.686,E2 -21457.686} C_VEL
LIN {X 0,Y 201.713,Z 605.308,A -85,B 0,C 180,E1 -21460.928,E2 -21460.928} C_VEL
LIN {X 0,Y 200.633,Z 607.801,A -85,B 0,C 180,E1 -21462.64,E2 -21462.64} C_VEL
LIN {X 0,Y 199.37,Z 610.562,A -85,B 0,C 180,E1 -21465.167,E2 -21465.167} C_VEL
LIN {X 0,Y 198.194,Z 612.652,A -85,B 0,C 180,E1 -21468.13,E2 -21468.13} C_VEL
LIN {X 0,Y 197.629,Z 613.527,A -85,B 0,C 180,E1 -21470.199,E2 -21470.199} C_VEL
LIN {X 0,Y 197.157,Z 613.847,A -85,B 0,C 180,E1 -21472.698,E2 -21472.698} C_VEL
LIN {X 0,Y 196.945,Z 613.423,A -85,B 0,C 180,E1 -21475.181,E2 -21475.181} C_VEL
LIN {X 0,Y 196.954,Z 612.268,A -85,B 0,C 180,E1 -21477.638,E2 -21477.638} C_VEL
LIN {X 0,Y 197.228,Z 610.377,A -85,B 0,C 180,E1 -21480.073,E2 -21480.073} C_VEL
LIN {X 0,Y 197.761,Z 607.485,A -85,B 0,C 180,E1 -21482.679,E2 -21482.679} C_VEL
LIN {X 0,Y 198.243,Z 604.331,A -85,B 0,C 180,E1 -21484.822,E2 -21484.822} C_VEL
LIN {X 0,Y 199.176,Z 598.832,A -85,B 0,C 180,E1 -21487.708,E2 -21487.708} C_VEL
LIN {X 0,Y 200.079,Z 593.673,A -85,B 0,C 180,E1 -21489.848,E2 -21489.848} C_VEL
LIN {X 0,Y 201.091,Z 588.398,A -85,B 0,C 180,E1 -21491.666,E2 -21491.666} C_VEL
LIN {X 0,Y 202.497,Z 580.439,A -85,B 0,C 180,E1 -21493.879,E2 -21493.879} C_VEL
LIN {X 0,Y 203.968,Z 572.02,A -85,B 0,C 180,E1 -21495.747,E2 -21495.747} C_VEL
LIN {X 0,Y 204.301,Z 567.745,A -85,B 0,C 180,E1 -21496.572,E2 -21496.572} C_VEL
LIN {X 0,Y 203.566,Z 559.392,A -85,B 0,C 180,E1 -21498.044,E2 -21498.044} C_VEL
LIN {X 0,Y 202.456,Z 550.006,A -85,B 0,C 180,E1 -21499.403,E2 -21499.403} C_VEL
LIN {X 0,Y 200.703,Z 539.292,A -85,B 0,C 180,E1 -21500.652,E2 -21500.652} C_VEL
LIN {X 0,Y 199.234,Z 531.844,A -85,B 0,C 180,E1 -21501.376,E2 -21501.376} C_VEL
LIN {X 0,Y 199.803,Z 525.999,A -85,B 0,C 180,E1 -21505.965,E2 -21505.965} C_VEL
LIN {X 0,Y 200.35,Z 520.345,A -85,B 0,C 180,E1 -21510.439,E2 -21510.439} C_VEL
LIN {X 0,Y 200.325,Z 520.344,A -85,B 0,C 180,E1 -21512.009,E2 -21512.009} C_VEL
LIN {X 0,Y 200.134,Z 520.37,A -85,B 0,C 180,E1 -21518.074,E2 -21518.074} C_VEL
LIN {X 0,Y 199.916,Z 520.396,A -85,B 0,C 180,E1 -21522.176,E2 -21522.176} C_VEL
LIN {X 0,Y 199.806,Z 520.409,A -85,B 0,C 180,E1 -21526.342,E2 -21526.342} C_VEL
LIN {X 0,Y 199.701,Z 520.421,A -85,B 0,C 180,E1 -21530.604,E2 -21530.604} C_VEL
LIN {X 0,Y 199.673,Z 520.423,A -85,B 0,C 180,E1 -21534.983,E2 -21534.983} C_VEL
LIN {X 0,Y 199.675,Z 520.424,A -85,B 0,C 180,E1 -21539.521,E2 -21539.521} C_VEL
LIN {X 0,Y 199.664,Z 520.426,A -85,B 0,C 180,E1 -21542.351,E2 -21542.351} C_VEL
LIN {X 0,Y 199.65,Z 520.426,A -85,B 0,C 180,E1 -21546.756,E2 -21546.756} C_VEL
LIN {X 0,Y 199.673,Z 520.423,A -85,B 0,C 180,E1 -21549.311,E2 -21549.311} C_VEL
LIN {X 0,Y 199.647,Z 520.423,A -85,B 0,C 180,E1 -21552.333,E2 -21552.333} C_VEL
LIN {X 0,Y 199.664,Z 520.423,A -85,B 0,C 180,E1 -21555.252,E2 -21555.252} C_VEL
LIN {X 0,Y 199.665,Z 520.428,A -85,B 0,C 180,E1 -21558.027,E2 -21558.027} C_VEL
LIN {X 0,Y 199.678,Z 520.42,A -85,B 0,C 180,E1 -21560.742,E2 -21560.742} C_VEL
LIN {X 0,Y 199.632,Z 520.427,A -85,B 0,C 180,E1 -21565.717,E2 -21565.717} C_VEL
LIN {X 0,Y 199.694,Z 520.424,A -85,B 0,C 180,E1 -21568.136,E2 -21568.136} C_VEL
LIN {X 0,Y 199.683,Z 520.419,A -85,B 0,C 180,E1 -21572.771,E2 -21572.771} C_VEL
LIN {X 0,Y 199.736,Z 520.416,A -85,B 0,C 180,E1 -21577.229,E2 -21577.229} C_VEL
LIN {X 0,Y 199.794,Z 520.407,A -85,B 0,C 180,E1 -21581.757,E2 -21581.757} C_VEL
LIN {X 0,Y 199.846,Z 520.405,A -85,B 0,C 180,E1 -21585.749,E2 -21585.749} C_VEL
LIN {X 0,Y 200.073,Z 520.374,A -85,B 0,C 180,E1 -21589.884,E2 -21589.884} C_VEL
LIN {X 0,Y 200.039,Z 520.38,A -85,B 0,C 180,E1 -21593.95,E2 -21593.95} C_VEL
LIN {X 0,Y 200.321,Z 520.337,A -85,B 0,C 180,E1 -21597.989,E2 -21597.989} C_VEL
LIN {X 0,Y 200.478,Z 520.32,A -85,B 0,C 180,E1 -21600,E2 -21600} C_VEL
LIN {X 0,Y 200.033,Z 520.381,A -85,B 0,C 180,E1 -21604.029,E2 -21604.029} C_VEL
LIN {X 0,Y 200.13,Z 520.368,A -85,B 0,C 180,E1 -21608.075,E2 -21608.075} C_VEL
LIN {X 0,Y 199.912,Z 520.395,A -85,B 0,C 180,E1 -21612.177,E2 -21612.177} C_VEL
LIN {X 0,Y 199.803,Z 520.408,A -85,B 0,C 180,E1 -21616.343,E2 -21616.343} C_VEL
LIN {X 0,Y 199.698,Z 520.421,A -85,B 0,C 180,E1 -21620.605,E2 -21620.605} C_VEL
LIN {X 0,Y 199.671,Z 520.426,A -85,B 0,C 180,E1 -21624.984,E2 -21624.984} C_VEL
LIN {X 0,Y 199.672,Z 520.428,A -85,B 0,C 180,E1 -21629.522,E2 -21629.522} C_VEL
LIN {X 0,Y 199.662,Z 520.426,A -85,B 0,C 180,E1 -21632.353,E2 -21632.353} C_VEL
LIN {X 0,Y 199.637,Z 520.428,A -85,B 0,C 180,E1 -21636.76,E2 -21636.76} C_VEL
LIN {X 0,Y 199.638,Z 520.43,A -85,B 0,C 180,E1 -21639.321,E2 -21639.321} C_VEL
LIN {X 0,Y 199.617,Z 520.432,A -85,B 0,C 180,E1 -21642.325,E2 -21642.325} C_VEL
LIN {X 0,Y 199.632,Z 520.431,A -85,B 0,C 180,E1 -21645.245,E2 -21645.245} C_VEL
LIN {X 0,Y 199.839,Z 520.405,A -85,B 0,C 180,E1 -21650.727,E2 -21650.727} C_VEL
LIN {X 0,Y 200.241,Z 520.455,A -85,B 0,C 180,E1 -21654.618,E2 -21654.618} C_VEL
LIN {X 0,Y 200.726,Z 523.058,A -85,B 0,C 180,E1 -21657.173,E2 -21657.173} C_VEL
LIN {X 0,Y 200.029,Z 526.556,A -85,B 0,C 180,E1 -21660.536,E2 -21660.536} C_VEL
LIN {X 0,Y 199.646,Z 528.173,A -85,B 0,C 180,E1 -21661.892,E2 -21661.892} C_VEL
LIN {X 0,Y 199.505,Z 536.565,A -85,B 0,C 180,E1 -21664.69,E2 -21664.69} C_VEL
LIN {X 0,Y 201.481,Z 549.765,A -85,B 0,C 180,E1 -21665.679,E2 -21665.679} C_VEL
LIN {X 0,Y 202.249,Z 559.792,A -85,B 0,C 180,E1 -21666.706,E2 -21666.706} C_VEL
LIN {X 0,Y 202.656,Z 568.583,A -85,B 0,C 180,E1 -21667.858,E2 -21667.858} C_VEL
LIN {X 0,Y 202.856,Z 577.407,A -85,B 0,C 180,E1 -21669.296,E2 -21669.296} C_VEL
LIN {X 0,Y 202.648,Z 586.265,A -85,B 0,C 180,E1 -21671.06,E2 -21671.06} C_VEL
LIN {X 0,Y 201.133,Z 595.174,A -85,B 0,C 180,E1 -21673.247,E2 -21673.247} C_VEL
LIN {X 0,Y 199.939,Z 601.611,A -85,B 0,C 180,E1 -21675.237,E2 -21675.237} C_VEL
LIN {X 0,Y 199.049,Z 606.953,A -85,B 0,C 180,E1 -21677.248,E2 -21677.248} C_VEL
LIN {X 0,Y 197.865,Z 610.208,A -85,B 0,C 180,E1 -21678.656,E2 -21678.656} C_VEL
LIN {X 0,Y 194.334,Z 614.655,A -85,B 0,C 180,E1 -21681.039,E2 -21681.039} C_VEL
LIN {X 0,Y 191.044,Z 618.235,A -85,B 0,C 180,E1 -21683.616,E2 -21683.616} C_VEL
LIN {X 0,Y 190.253,Z 620.005,A -85,B 0,C 180,E1 -21685.287,E2 -21685.287} C_VEL
LIN {X 0,Y 190.242,Z 622.146,A -85,B 0,C 180,E1 -21687.884,E2 -21687.884} C_VEL
LIN {X 0,Y 190.366,Z 623.251,A -85,B 0,C 180,E1 -21690.001,E2 -21690.001} C_VEL
LIN {X 0,Y 190.226,Z 623.852,A -85,B 0,C 180,E1 -21692.118,E2 -21692.118} C_VEL
LIN {X 0,Y 190.236,Z 623.983,A -85,B 0,C 180,E1 -21694.238,E2 -21694.238} C_VEL
LIN {X 0,Y 190.427,Z 623.606,A -85,B 0,C 180,E1 -21696.358,E2 -21696.358} C_VEL
LIN {X 0,Y 190.776,Z 622.65,A -85,B 0,C 180,E1 -21698.475,E2 -21698.475} C_VEL
LIN {X 0,Y 191.388,Z 621.207,A -85,B 0,C 180,E1 -21700.581,E2 -21700.581} C_VEL
LIN {X 0,Y 192.779,Z 618.104,A -85,B 0,C 180,E1 -21703.709,E2 -21703.709} C_VEL
LIN {X 0,Y 193.573,Z 616.442,A -85,B 0,C 180,E1 -21704.993,E2 -21704.993} C_VEL
LIN {X 0,Y 194.829,Z 616.43,A -85,B 0,C 180,E1 -21706.774,E2 -21706.774} C_VEL
LIN {X 0,Y 198.678,Z 615.044,A -85,B 0,C 180,E1 -21710.717,E2 -21710.717} C_VEL
LIN {X 0,Y 201.086,Z 613.844,A -85,B 0,C 180,E1 -21712.611,E2 -21712.611} C_VEL
LIN {X 0,Y 205.232,Z 611.201,A -85,B 0,C 180,E1 -21715.345,E2 -21715.345} C_VEL
LIN {X 0,Y 210.129,Z 607.565,A -85,B 0,C 180,E1 -21717.922,E2 -21717.922} C_VEL
LIN {X 0,Y 213.39,Z 604.679,A -85,B 0,C 180,E1 -21719.607,E2 -21719.607} C_VEL
LIN {X 0,Y 216.765,Z 600.306,A -85,B 0,C 180,E1 -21722.171,E2 -21722.171} C_VEL
LIN {X 0,Y 219.722,Z 595.275,A -85,B 0,C 180,E1 -21725.153,E2 -21725.153} C_VEL
LIN {X 0,Y 222.009,Z 590.622,A -85,B 0,C 180,E1 -21728.119,E2 -21728.119} C_VEL
LIN {X 0,Y 222.559,Z 589.234,A -85,B 0,C 180,E1 -21729.167,E2 -21729.167} C_VEL
LIN {X 0,Y 222.99,Z 587.582,A -85,B 0,C 180,E1 -21730.851,E2 -21730.851} C_VEL
LIN {X 0,Y 223.024,Z 585.789,A -85,B 0,C 180,E1 -21733.891,E2 -21733.891} C_VEL
LIN {X 0,Y 223.161,Z 584.919,A -85,B 0,C 180,E1 -21736.415,E2 -21736.415} C_VEL
LIN {X 0,Y 223.295,Z 584.75,A -85,B 0,C 180,E1 -21739.06,E2 -21739.06} C_VEL
LIN {X 0,Y 223.385,Z 585.333,A -85,B 0,C 180,E1 -21741.864,E2 -21741.864} C_VEL
LIN {X 0,Y 223.359,Z 586.024,A -85,B 0,C 180,E1 -21743.285,E2 -21743.285} C_VEL
LIN {X 0,Y 223.005,Z 587.59,A -85,B 0,C 180,E1 -21745.44,E2 -21745.44} C_VEL
LIN {X 0,Y 222.183,Z 589.458,A -85,B 0,C 180,E1 -21747.47,E2 -21747.47} C_VEL
LIN {X 0,Y 221.135,Z 591.649,A -85,B 0,C 180,E1 -21749.436,E2 -21749.436} C_VEL
LIN {X 0,Y 220.15,Z 592.809,A -85,B 0,C 180,E1 -21750.342,E2 -21750.342} C_VEL
LIN {X 0,Y 214.657,Z 596.964,A -85,B 0,C 180,E1 -21752.718,E2 -21752.718} C_VEL
LIN {X 0,Y 211.209,Z 599.233,A -85,B 0,C 180,E1 -21754.369,E2 -21754.369} C_VEL
LIN {X 0,Y 208.016,Z 601.032,A -85,B 0,C 180,E1 -21756.082,E2 -21756.082} C_VEL
LIN {X 0,Y 202.356,Z 603.172,A -85,B 0,C 180,E1 -21759.677,E2 -21759.677} C_VEL
LIN {X 0,Y 199.961,Z 603.699,A -85,B 0,C 180,E1 -21761.56,E2 -21761.56} C_VEL
LIN {X 0,Y 197.795,Z 603.742,A -85,B 0,C 180,E1 -21763.486,E2 -21763.486} C_VEL
LIN {X 0,Y 194.21,Z 602.559,A -85,B 0,C 180,E1 -21767.46,E2 -21767.46} C_VEL
LIN {X 0,Y 192.985,Z 601.388,A -85,B 0,C 180,E1 -21769.509,E2 -21769.509} C_VEL
LIN {X 0,Y 191.777,Z 598.768,A -85,B 0,C 180,E1 -21772.631,E2 -21772.631} C_VEL
LIN {X 0,Y 191.072,Z 595.06,A -85,B 0,C 180,E1 -21775.781,E2 -21775.781} C_VEL
LIN {X 0,Y 190.654,Z 590.174,A -85,B 0,C 180,E1 -21778.944,E2 -21778.944} C_VEL
LIN {X 0,Y 190.755,Z 585.16,A -85,B 0,C 180,E1 -21781.584,E2 -21781.584} C_VEL
LIN {X 0,Y 190.941,Z 578.979,A -85,B 0,C 180,E1 -21784.222,E2 -21784.222} C_VEL
LIN {X 0,Y 191.403,Z 570.895,A -85,B 0,C 180,E1 -21787.046,E2 -21787.046} C_VEL
LIN {X 0,Y 192.033,Z 561.101,A -85,B 0,C 180,E1 -21789.745,E2 -21789.745} C_VEL
LIN {X 0,Y 192.587,Z 553.016,A -85,B 0,C 180,E1 -21791.579,E2 -21791.579} C_VEL
LIN {X 0,Y 193.293,Z 543.297,A -85,B 0,C 180,E1 -21793.403,E2 -21793.403} C_VEL
LIN {X 0,Y 192.817,Z 538.671,A -85,B 0,C 180,E1 -21794.108,E2 -21794.108} C_VEL
LIN {X 0,Y 191.594,Z 529.62,A -85,B 0,C 180,E1 -21795.287,E2 -21795.287} C_VEL
LIN {X 0,Y 193.12,Z 532.781,A -85,B 0,C 180,E1 -21798.922,E2 -21798.922} C_VEL
LIN {X 0,Y 195.137,Z 536.372,A -85,B 0,C 180,E1 -21799.871,E2 -21799.871} C_VEL
LIN {X 0,Y 196.685,Z 538.566,A -85,B 0,C 180,E1 -21800.526,E2 -21800.526} C_VEL
LIN {X 0,Y 201.017,Z 546.25,A -85,B 0,C 180,E1 -21802.618,E2 -21802.618} C_VEL
LIN {X 0,Y 202.862,Z 550.953,A -85,B 0,C 180,E1 -21803.75,E2 -21803.75} C_VEL
LIN {X 0,Y 204.644,Z 560.073,A -85,B 0,C 180,E1 -21805.695,E2 -21805.695} C_VEL
LIN {X 0,Y 205.497,Z 569.299,A -85,B 0,C 180,E1 -21807.773,E2 -21807.773} C_VEL
LIN {X 0,Y 205.321,Z 578.034,A -85,B 0,C 180,E1 -21809.931,E2 -21809.931} C_VEL
LIN {X 0,Y 204.625,Z 581.475,A -85,B 0,C 180,E1 -21810.834,E2 -21810.834} C_VEL
LIN {X 0,Y 202.348,Z 588.099,A -85,B 0,C 180,E1 -21812.619,E2 -21812.619} C_VEL
LIN {X 0,Y 199.739,Z 594.839,A -85,B 0,C 180,E1 -21814.867,E2 -21814.867} C_VEL
LIN {X 0,Y 197.409,Z 600.409,A -85,B 0,C 180,E1 -21817.245,E2 -21817.245} C_VEL
LIN {X 0,Y 195.638,Z 604.38,A -85,B 0,C 180,E1 -21819.404,E2 -21819.404} C_VEL
LIN {X 0,Y 193.857,Z 608.101,A -85,B 0,C 180,E1 -21821.994,E2 -21821.994} C_VEL
LIN {X 0,Y 192.847,Z 610.069,A -85,B 0,C 180,E1 -21823.822,E2 -21823.822} C_VEL
LIN {X 0,Y 191.363,Z 612.714,A -85,B 0,C 180,E1 -21827.267,E2 -21827.267} C_VEL
LIN {X 0,Y 190.326,Z 613.918,A -85,B 0,C 180,E1 -21831.115,E2 -21831.115} C_VEL
LIN {X 0,Y 189.878,Z 613.699,A -85,B 0,C 180,E1 -21834.518,E2 -21834.518} C_VEL
LIN {X 0,Y 189.912,Z 611.838,A -85,B 0,C 180,E1 -21838.338,E2 -21838.338} C_VEL
LIN {X 0,Y 190.375,Z 609.191,A -85,B 0,C 180,E1 -21841.319,E2 -21841.319} C_VEL
LIN {X 0,Y 191.166,Z 604.411,A -85,B 0,C 180,E1 -21844.988,E2 -21844.988} C_VEL
LIN {X 0,Y 192.166,Z 598.694,A -85,B 0,C 180,E1 -21848.055,E2 -21848.055} C_VEL
LIN {X 0,Y 193.202,Z 593.144,A -85,B 0,C 180,E1 -21850.392,E2 -21850.392} C_VEL
LIN {X 0,Y 194.539,Z 586.466,A -85,B 0,C 180,E1 -21852.659,E2 -21852.659} C_VEL
LIN {X 0,Y 195.994,Z 578.524,A -85,B 0,C 180,E1 -21854.832,E2 -21854.832} C_VEL
LIN {X 0,Y 197.354,Z 570.388,A -85,B 0,C 180,E1 -21856.615,E2 -21856.615} C_VEL
LIN {X 0,Y 196.73,Z 560.618,A -85,B 0,C 180,E1 -21858.445,E2 -21858.445} C_VEL
LIN {X 0,Y 195.669,Z 551.212,A -85,B 0,C 180,E1 -21859.88,E2 -21859.88} C_VEL
LIN {X 0,Y 194.037,Z 541.102,A -85,B 0,C 180,E1 -21861.131,E2 -21861.131} C_VEL
LIN {X 0,Y 192.267,Z 532.006,A -85,B 0,C 180,E1 -21862.054,E2 -21862.054} C_VEL
LIN {X 0,Y 192.76,Z 527.33,A -85,B 0,C 180,E1 -21865.817,E2 -21865.817} C_VEL
LIN {X 0,Y 193.358,Z 521.499,A -85,B 0,C 180,E1 -21870.52,E2 -21870.52} C_VEL
LIN {X 0,Y 193.305,Z 521.219,A -85,B 0,C 180,E1 -21871.041,E2 -21871.041} C_VEL
LIN {X 0,Y 193.081,Z 521.248,A -85,B 0,C 180,E1 -21878.371,E2 -21878.371} C_VEL
LIN {X 0,Y 192.855,Z 521.275,A -85,B 0,C 180,E1 -21882.629,E2 -21882.629} C_VEL
LIN {X 0,Y 192.759,Z 521.285,A -85,B 0,C 180,E1 -21886.957,E2 -21886.957} C_VEL
LIN {X 0,Y 192.637,Z 521.299,A -85,B 0,C 180,E1 -21891.396,E2 -21891.396} C_VEL
LIN {X 0,Y 192.664,Z 521.297,A -85,B 0,C 180,E1 -21894.224,E2 -21894.224} C_VEL
LIN {X 0,Y 192.65,Z 521.299,A -85,B 0,C 180,E1 -21898.891,E2 -21898.891} C_VEL
LIN {X 0,Y 192.6,Z 521.304,A -85,B 0,C 180,E1 -21903.184,E2 -21903.184} C_VEL
LIN {X 0,Y 192.597,Z 521.307,A -85,B 0,C 180,E1 -21908.34,E2 -21908.34} C_VEL
LIN {X 0,Y 192.599,Z 521.301,A -85,B 0,C 180,E1 -21913.892,E2 -21913.892} C_VEL
LIN {X 0,Y 192.582,Z 521.306,A -85,B 0,C 180,E1 -21918.937,E2 -21918.937} C_VEL
LIN {X 0,Y 192.617,Z 521.295,A -85,B 0,C 180,E1 -21923.388,E2 -21923.388} C_VEL
LIN {X 0,Y 192.603,Z 521.303,A -85,B 0,C 180,E1 -21927.06,E2 -21927.06} C_VEL
LIN {X 0,Y 192.658,Z 521.298,A -85,B 0,C 180,E1 -21931.691,E2 -21931.691} C_VEL
LIN {X 0,Y 192.704,Z 521.293,A -85,B 0,C 180,E1 -21936.348,E2 -21936.348} C_VEL
LIN {X 0,Y 192.73,Z 521.286,A -85,B 0,C 180,E1 -21941.457,E2 -21941.457} C_VEL
LIN {X 0,Y 192.77,Z 521.284,A -85,B 0,C 180,E1 -21945.214,E2 -21945.214} C_VEL
LIN {X 0,Y 193.018,Z 521.25,A -85,B 0,C 180,E1 -21949.51,E2 -21949.51} C_VEL
LIN {X 0,Y 193.003,Z 521.258,A -85,B 0,C 180,E1 -21953.728,E2 -21953.728} C_VEL
LIN {X 0,Y 193.263,Z 521.216,A -85,B 0,C 180,E1 -21957.916,E2 -21957.916} C_VEL
LIN {X 0,Y 193.441,Z 521.196,A -85,B 0,C 180,E1 -21960,E2 -21960} C_VEL
LIN {X 0,Y 192.979,Z 521.259,A -85,B 0,C 180,E1 -21964.177,E2 -21964.177} C_VEL
LIN {X 0,Y 193.077,Z 521.246,A -85,B 0,C 180,E1 -21968.372,E2 -21968.372} C_VEL
LIN {X 0,Y 192.851,Z 521.273,A -85,B 0,C 180,E1 -21972.63,E2 -21972.63} C_VEL
LIN {X 0,Y 192.755,Z 521.285,A -85,B 0,C 180,E1 -21976.959,E2 -21976.959} C_VEL
LIN {X 0,Y 192.635,Z 521.303,A -85,B 0,C 180,E1 -21981.397,E2 -21981.397} C_VEL
LIN {X 0,Y 192.662,Z 521.299,A -85,B 0,C 180,E1 -21984.225,E2 -21984.225} C_VEL
LIN {X 0,Y 192.647,Z 521.3,A -85,B 0,C 180,E1 -21988.892,E2 -21988.892} C_VEL
LIN {X 0,Y 192.598,Z 521.307,A -85,B 0,C 180,E1 -21993.186,E2 -21993.186} C_VEL
LIN {X 0,Y 192.607,Z 521.304,A -85,B 0,C 180,E1 -21996.608,E2 -21996.608} C_VEL
LIN {X 0,Y 192.545,Z 521.314,A -85,B 0,C 180,E1 -22001.072,E2 -22001.072} C_VEL
LIN {X 0,Y 192.585,Z 521.308,A -85,B 0,C 180,E1 -22006.104,E2 -22006.104} C_VEL
LIN {X 0,Y 192.867,Z 521.275,A -85,B 0,C 180,E1 -22011.724,E2 -22011.724} C_VEL
LIN {X 0,Y 193.26,Z 521.326,A -85,B 0,C 180,E1 -22015.151,E2 -22015.151} C_VEL
LIN {X 0,Y 193.603,Z 523.15,A -85,B 0,C 180,E1 -22017.01,E2 -22017.01} C_VEL
LIN {X 0,Y 192.917,Z 526.767,A -85,B 0,C 180,E1 -22020.544,E2 -22020.544} C_VEL
LIN {X 0,Y 192.628,Z 536.55,A -85,B 0,C 180,E1 -22024,E2 -22024} C_VEL
LIN {X 0,Y 194.624,Z 549.739,A -85,B 0,C 180,E1 -22025.039,E2 -22025.039} C_VEL
LIN {X 0,Y 195.382,Z 560.251,A -85,B 0,C 180,E1 -22026.164,E2 -22026.164} C_VEL
LIN {X 0,Y 195.77,Z 568.909,A -85,B 0,C 180,E1 -22027.356,E2 -22027.356} C_VEL
LIN {X 0,Y 195.905,Z 577.77,A -85,B 0,C 180,E1 -22028.865,E2 -22028.865} C_VEL
LIN {X 0,Y 195.615,Z 587.28,A -85,B 0,C 180,E1 -22030.863,E2 -22030.863} C_VEL
LIN {X 0,Y 193.975,Z 595.949,A -85,B 0,C 180,E1 -22033.152,E2 -22033.152} C_VEL
LIN {X 0,Y 192.783,Z 602.227,A -85,B 0,C 180,E1 -22035.216,E2 -22035.216} C_VEL
LIN {X 0,Y 191.88,Z 607.44,A -85,B 0,C 180,E1 -22037.306,E2 -22037.306} C_VEL
LIN {X 0,Y 191.203,Z 611.768,A -85,B 0,C 180,E1 -22039.411,E2 -22039.411} C_VEL
LIN {X 0,Y 190.496,Z 616.844,A -85,B 0,C 180,E1 -22042.582,E2 -22042.582} C_VEL
LIN {X 0,Y 190.253,Z 620.005,A -85,B 0,C 180,E1 -22045.287,E2 -22045.287} C_VEL
LIN {X 0,Y 189.894,Z 621.113,A -85,B 0,C 180,E1 -22046.423,E2 -22046.423} C_VEL
LIN {X 0,Y 188.499,Z 622.416,A -85,B 0,C 180,E1 -22048.128,E2 -22048.128} C_VEL
LIN {X 0,Y 185.31,Z 623.665,A -85,B 0,C 180,E1 -22051.012,E2 -22051.012} C_VEL
LIN {X 0,Y 183.422,Z 623.902,A -85,B 0,C 180,E1 -22053.437,E2 -22053.437} C_VEL
LIN {X 0,Y 183.169,Z 623.777,A -85,B 0,C 180,E1 -22054.685,E2 -22054.685} C_VEL
LIN {X 0,Y 183.375,Z 623.462,A -85,B 0,C 180,E1 -22056.603,E2 -22056.603} C_VEL
LIN {X 0,Y 183.759,Z 622.57,A -85,B 0,C 180,E1 -22058.801,E2 -22058.801} C_VEL
LIN {X 0,Y 184.407,Z 621.207,A -85,B 0,C 180,E1 -22060.986,E2 -22060.986} C_VEL
LIN {X 0,Y 185.896,Z 618.198,A -85,B 0,C 180,E1 -22064.227,E2 -22064.227} C_VEL
LIN {X 0,Y 187.104,Z 615.906,A -85,B 0,C 180,E1 -22066.084,E2 -22066.084} C_VEL
LIN {X 0,Y 189.848,Z 615.681,A -85,B 0,C 180,E1 -22069.463,E2 -22069.463} C_VEL
LIN {X 0,Y 192.061,Z 615.097,A -85,B 0,C 180,E1 -22071.466,E2 -22071.466} C_VEL
LIN {X 0,Y 197.318,Z 612.626,A -85,B 0,C 180,E1 -22075.305,E2 -22075.305} C_VEL
LIN {X 0,Y 202.176,Z 609.729,A -85,B 0,C 180,E1 -22077.989,E2 -22077.989} C_VEL
LIN {X 0,Y 207.354,Z 605.978,A -85,B 0,C 180,E1 -22080.559,E2 -22080.559} C_VEL
LIN {X 0,Y 211.061,Z 601.845,A -85,B 0,C 180,E1 -22083.318,E2 -22083.318} C_VEL
LIN {X 0,Y 214.118,Z 597.537,A -85,B 0,C 180,E1 -22086.216,E2 -22086.216} C_VEL
LIN {X 0,Y 216.282,Z 594.038,A -85,B 0,C 180,E1 -22088.752,E2 -22088.752} C_VEL
LIN {X 0,Y 217.025,Z 592.376,A -85,B 0,C 180,E1 -22090.367,E2 -22090.367} C_VEL
LIN {X 0,Y 217.265,Z 590.682,A -85,B 0,C 180,E1 -22092.79,E2 -22092.79} C_VEL
LIN {X 0,Y 217.425,Z 589.6,A -85,B 0,C 180,E1 -22095.328,E2 -22095.328} C_VEL
LIN {X 0,Y 217.582,Z 589.123,A -85,B 0,C 180,E1 -22097.981,E2 -22097.981} C_VEL
LIN {X 0,Y 217.713,Z 589.343,A -85,B 0,C 180,E1 -22100.783,E2 -22100.783} C_VEL
LIN {X 0,Y 217.655,Z 589.683,A -85,B 0,C 180,E1 -22102.157,E2 -22102.157} C_VEL
LIN {X 0,Y 217.204,Z 590.813,A -85,B 0,C 180,E1 -22104.379,E2 -22104.379} C_VEL
LIN {X 0,Y 216.425,Z 592.428,A -85,B 0,C 180,E1 -22106.493,E2 -22106.493} C_VEL
LIN {X 0,Y 215.24,Z 594.116,A -85,B 0,C 180,E1 -22108.505,E2 -22108.505} C_VEL
LIN {X 0,Y 214.291,Z 595.187,A -85,B 0,C 180,E1 -22109.446,E2 -22109.446} C_VEL
LIN {X 0,Y 208.585,Z 598.961,A -85,B 0,C 180,E1 -22111.855,E2 -22111.855} C_VEL
LIN {X 0,Y 201.652,Z 602.312,A -85,B 0,C 180,E1 -22115.278,E2 -22115.278} C_VEL
LIN {X 0,Y 198.59,Z 603.435,A -85,B 0,C 180,E1 -22117.09,E2 -22117.09} C_VEL
LIN {X 0,Y 195.78,Z 604.053,A -85,B 0,C 180,E1 -22118.963,E2 -22118.963} C_VEL
LIN {X 0,Y 191.034,Z 604.103,A -85,B 0,C 180,E1 -22122.884,E2 -22122.884} C_VEL
LIN {X 0,Y 189.1,Z 603.539,A -85,B 0,C 180,E1 -22124.921,E2 -22124.921} C_VEL
LIN {X 0,Y 187.3,Z 602.47,A -85,B 0,C 180,E1 -22126.989,E2 -22126.989} C_VEL
LIN {X 0,Y 185.115,Z 599.242,A -85,B 0,C 180,E1 -22131.265,E2 -22131.265} C_VEL
LIN {X 0,Y 184.239,Z 595.598,A -85,B 0,C 180,E1 -22134.528,E2 -22134.528} C_VEL
LIN {X 0,Y 183.723,Z 590.804,A -85,B 0,C 180,E1 -22137.808,E2 -22137.808} C_VEL
LIN {X 0,Y 183.706,Z 585.827,A -85,B 0,C 180,E1 -22140.548,E2 -22140.548} C_VEL
LIN {X 0,Y 183.898,Z 579.798,A -85,B 0,C 180,E1 -22143.286,E2 -22143.286} C_VEL
LIN {X 0,Y 184.203,Z 572.717,A -85,B 0,C 180,E1 -22145.945,E2 -22145.945} C_VEL
LIN {X 0,Y 184.795,Z 563.482,A -85,B 0,C 180,E1 -22148.75,E2 -22148.75} C_VEL
LIN {X 0,Y 185.409,Z 554.507,A -85,B 0,C 180,E1 -22150.925,E2 -22150.925} C_VEL
LIN {X 0,Y 186.144,Z 545.046,A -85,B 0,C 180,E1 -22152.816,E2 -22152.816} C_VEL
LIN {X 0,Y 186.232,Z 541.989,A -85,B 0,C 180,E1 -22153.365,E2 -22153.365} C_VEL
LIN {X 0,Y 184.775,Z 531.815,A -85,B 0,C 180,E1 -22154.806,E2 -22154.806} C_VEL
LIN {X 0,Y 185.384,Z 533.047,A -85,B 0,C 180,E1 -22156.307,E2 -22156.307} C_VEL
LIN {X 0,Y 188.116,Z 537.157,A -85,B 0,C 180,E1 -22157.703,E2 -22157.703} C_VEL
LIN {X 0,Y 189.361,Z 538.75,A -85,B 0,C 180,E1 -22158.284,E2 -22158.284} C_VEL
LIN {X 0,Y 191.817,Z 542.723,A -85,B 0,C 180,E1 -22159.555,E2 -22159.555} C_VEL
LIN {X 0,Y 196.078,Z 550.866,A -85,B 0,C 180,E1 -22161.97,E2 -22161.97} C_VEL
LIN {X 0,Y 197.56,Z 555.048,A -85,B 0,C 180,E1 -22163.036,E2 -22163.036} C_VEL
LIN {X 0,Y 199.066,Z 564.937,A -85,B 0,C 180,E1 -22165.345,E2 -22165.345} C_VEL
LIN {X 0,Y 199.35,Z 572.721,A -85,B 0,C 180,E1 -22167.278,E2 -22167.278} C_VEL
LIN {X 0,Y 198.92,Z 580.106,A -85,B 0,C 180,E1 -22169.284,E2 -22169.284} C_VEL
LIN {X 0,Y 198.203,Z 582.991,A -85,B 0,C 180,E1 -22170.047,E2 -22170.047} C_VEL
LIN {X 0,Y 195.08,Z 591.254,A -85,B 0,C 180,E1 -22172.476,E2 -22172.476} C_VEL
LIN {X 0,Y 192.489,Z 597.249,A -85,B 0,C 180,E1 -22174.765,E2 -22174.765} C_VEL
LIN {X 0,Y 190.063,Z 602.518,A -85,B 0,C 180,E1 -22177.342,E2 -22177.342} C_VEL
LIN {X 0,Y 188.439,Z 605.803,A -85,B 0,C 180,E1 -22179.348,E2 -22179.348} C_VEL
LIN {X 0,Y 187.107,Z 608.424,A -85,B 0,C 180,E1 -22181.302,E2 -22181.302} C_VEL
LIN {X 0,Y 185.611,Z 611.102,A -85,B 0,C 180,E1 -22183.992,E2 -22183.992} C_VEL
LIN {X 0,Y 184.468,Z 612.927,A -85,B 0,C 180,E1 -22186.702,E2 -22186.702} C_VEL
LIN {X 0,Y 183.464,Z 614.034,A -85,B 0,C 180,E1 -22190.009,E2 -22190.009} C_VEL
LIN {X 0,Y 183.034,Z 614.231,A -85,B 0,C 180,E1 -22192.094,E2 -22192.094} C_VEL
LIN {X 0,Y 182.761,Z 613.76,A -85,B 0,C 180,E1 -22194.772,E2 -22194.772} C_VEL
LIN {X 0,Y 182.763,Z 612.318,A -85,B 0,C 180,E1 -22197.779,E2 -22197.779} C_VEL
LIN {X 0,Y 183.024,Z 610.616,A -85,B 0,C 180,E1 -22200.052,E2 -22200.052} C_VEL
LIN {X 0,Y 183.517,Z 607.921,A -85,B 0,C 180,E1 -22202.64,E2 -22202.64} C_VEL
LIN {X 0,Y 184.113,Z 604.453,A -85,B 0,C 180,E1 -22205.171,E2 -22205.171} C_VEL
LIN {X 0,Y 185.118,Z 598.842,A -85,B 0,C 180,E1 -22208.273,E2 -22208.273} C_VEL
LIN {X 0,Y 186.171,Z 593.296,A -85,B 0,C 180,E1 -22210.692,E2 -22210.692} C_VEL
LIN {X 0,Y 187.218,Z 588.243,A -85,B 0,C 180,E1 -22212.522,E2 -22212.522} C_VEL
LIN {X 0,Y 188.526,Z 581.307,A -85,B 0,C 180,E1 -22214.596,E2 -22214.596} C_VEL
LIN {X 0,Y 189.915,Z 574.086,A -85,B 0,C 180,E1 -22216.353,E2 -22216.353} C_VEL
LIN {X 0,Y 190.429,Z 568.856,A -85,B 0,C 180,E1 -22217.476,E2 -22217.476} C_VEL
LIN {X 0,Y 189.792,Z 560.614,A -85,B 0,C 180,E1 -22219.059,E2 -22219.059} C_VEL
LIN {X 0,Y 188.667,Z 551.248,A -85,B 0,C 180,E1 -22220.55,E2 -22220.55} C_VEL
LIN {X 0,Y 187.192,Z 541.82,A -85,B 0,C 180,E1 -22221.769,E2 -22221.769} C_VEL
LIN {X 0,Y 185.328,Z 532.168,A -85,B 0,C 180,E1 -22222.783,E2 -22222.783} C_VEL
LIN {X 0,Y 185.979,Z 526.031,A -85,B 0,C 180,E1 -22227.833,E2 -22227.833} C_VEL
LIN {X 0,Y 186.285,Z 522.143,A -85,B 0,C 180,E1 -22231.08,E2 -22231.08} C_VEL
LIN {X 0,Y 185.971,Z 522.134,A -85,B 0,C 180,E1 -22236.509,E2 -22236.509} C_VEL
LIN {X 0,Y 185.944,Z 522.136,A -85,B 0,C 180,E1 -22240.671,E2 -22240.671} C_VEL
LIN {X 0,Y 185.725,Z 522.161,A -85,B 0,C 180,E1 -22245.359,E2 -22245.359} C_VEL
LIN {X 0,Y 185.608,Z 522.175,A -85,B 0,C 180,E1 -22249.923,E2 -22249.923} C_VEL
LIN {X 0,Y 185.601,Z 522.177,A -85,B 0,C 180,E1 -22254.661,E2 -22254.661} C_VEL
LIN {X 0,Y 185.579,Z 522.18,A -85,B 0,C 180,E1 -22259.492,E2 -22259.492} C_VEL
LIN {X 0,Y 185.52,Z 522.184,A -85,B 0,C 180,E1 -22264.626,E2 -22264.626} C_VEL
LIN {X 0,Y 185.543,Z 522.184,A -85,B 0,C 180,E1 -22267.303,E2 -22267.303} C_VEL
LIN {X 0,Y 185.527,Z 522.183,A -85,B 0,C 180,E1 -22270.745,E2 -22270.745} C_VEL
LIN {X 0,Y 185.563,Z 522.182,A -85,B 0,C 180,E1 -22276.02,E2 -22276.02} C_VEL
LIN {X 0,Y 185.54,Z 522.185,A -85,B 0,C 180,E1 -22279.914,E2 -22279.914} C_VEL
LIN {X 0,Y 185.558,Z 522.173,A -85,B 0,C 180,E1 -22282.699,E2 -22282.699} C_VEL
LIN {X 0,Y 185.539,Z 522.187,A -85,B 0,C 180,E1 -22287.974,E2 -22287.974} C_VEL
LIN {X 0,Y 185.578,Z 522.179,A -85,B 0,C 180,E1 -22290.576,E2 -22290.576} C_VEL
LIN {X 0,Y 185.585,Z 522.178,A -85,B 0,C 180,E1 -22295.382,E2 -22295.382} C_VEL
LIN {X 0,Y 185.605,Z 522.174,A -85,B 0,C 180,E1 -22300.075,E2 -22300.075} C_VEL
LIN {X 0,Y 185.722,Z 522.162,A -85,B 0,C 180,E1 -22304.639,E2 -22304.639} C_VEL
LIN {X 0,Y 185.94,Z 522.131,A -85,B 0,C 180,E1 -22309.328,E2 -22309.328} C_VEL
LIN {X 0,Y 185.967,Z 522.133,A -85,B 0,C 180,E1 -22313.49,E2 -22313.49} C_VEL
LIN {X 0,Y 186.207,Z 522.095,A -85,B 0,C 180,E1 -22317.837,E2 -22317.837} C_VEL
LIN {X 0,Y 186.405,Z 522.072,A -85,B 0,C 180,E1 -22320,E2 -22320} C_VEL
LIN {X 0,Y 185.927,Z 522.137,A -85,B 0,C 180,E1 -22324.335,E2 -22324.335} C_VEL
LIN {X 0,Y 186.027,Z 522.124,A -85,B 0,C 180,E1 -22328.692,E2 -22328.692} C_VEL
LIN {X 0,Y 185.763,Z 522.157,A -85,B 0,C 180,E1 -22333.12,E2 -22333.12} C_VEL
LIN {X 0,Y 185.688,Z 522.169,A -85,B 0,C 180,E1 -22337.625,E2 -22337.625} C_VEL
LIN {X 0,Y 185.595,Z 522.18,A -85,B 0,C 180,E1 -22342.251,E2 -22342.251} C_VEL
LIN {X 0,Y 185.56,Z 522.185,A -85,B 0,C 180,E1 -22347.032,E2 -22347.032} C_VEL
LIN {X 0,Y 185.576,Z 522.184,A -85,B 0,C 180,E1 -22349.493,E2 -22349.493} C_VEL
LIN {X 0,Y 185.517,Z 522.187,A -85,B 0,C 180,E1 -22354.628,E2 -22354.628} C_VEL
LIN {X 0,Y 185.541,Z 522.185,A -85,B 0,C 180,E1 -22357.305,E2 -22357.305} C_VEL
LIN {X 0,Y 185.5,Z 522.19,A -85,B 0,C 180,E1 -22360.737,E2 -22360.737} C_VEL
LIN {X 0,Y 185.547,Z 522.185,A -85,B 0,C 180,E1 -22366.027,E2 -22366.027} C_VEL
LIN {X 0,Y 185.667,Z 522.171,A -85,B 0,C 180,E1 -22369.948,E2 -22369.948} C_VEL
LIN {X 0,Y 186.309,Z 522.13,A -85,B 0,C 180,E1 -22375.68,E2 -22375.68} C_VEL
LIN {X 0,Y 186.223,Z 525.044,A -85,B 0,C 180,E1 -22378.742,E2 -22378.742} C_VEL
LIN {X 0,Y 186.15,Z 525.698,A -85,B 0,C 180,E1 -22379.202,E2 -22379.202} C_VEL
LIN {X 0,Y 185.799,Z 536.855,A -85,B 0,C 180,E1 -22383.304,E2 -22383.304} C_VEL
LIN {X 0,Y 187.784,Z 549.811,A -85,B 0,C 180,E1 -22384.373,E2 -22384.373} C_VEL
LIN {X 0,Y 188.458,Z 559.077,A -85,B 0,C 180,E1 -22385.394,E2 -22385.394} C_VEL
LIN {X 0,Y 188.866,Z 568.416,A -85,B 0,C 180,E1 -22386.712,E2 -22386.712} C_VEL
LIN {X 0,Y 188.971,Z 576.75,A -85,B 0,C 180,E1 -22388.168,E2 -22388.168} C_VEL
LIN {X 0,Y 188.735,Z 586.105,A -85,B 0,C 180,E1 -22390.166,E2 -22390.166} C_VEL
LIN {X 0,Y 187.184,Z 594.97,A -85,B 0,C 180,E1 -22392.521,E2 -22392.521} C_VEL
LIN {X 0,Y 185.888,Z 601.369,A -85,B 0,C 180,E1 -22394.655,E2 -22394.655} C_VEL
LIN {X 0,Y 184.936,Z 606.693,A -85,B 0,C 180,E1 -22396.821,E2 -22396.821} C_VEL
LIN {X 0,Y 184.196,Z 611.121,A -85,B 0,C 180,E1 -22399.003,E2 -22399.003} C_VEL
LIN {X 0,Y 183.46,Z 616.293,A -85,B 0,C 180,E1 -22402.296,E2 -22402.296} C_VEL
LIN {X 0,Y 183.165,Z 619.735,A -85,B 0,C 180,E1 -22405.287,E2 -22405.287} C_VEL
LIN {X 0,Y 183.15,Z 621.762,A -85,B 0,C 180,E1 -22407.802,E2 -22407.802} C_VEL
LIN {X 0,Y 183.266,Z 622.944,A -85,B 0,C 180,E1 -22410.001,E2 -22410.001} C_VEL
LIN {X 0,Y 183.141,Z 623.824,A -85,B 0,C 180,E1 -22413.852,E2 -22413.852} C_VEL
LIN {X 0,Y 183.169,Z 623.777,A -85,B 0,C 180,E1 -22414.685,E2 -22414.685} C_VEL
LIN {X 0,Y 182.67,Z 623.474,A -85,B 0,C 180,E1 -22416.527,E2 -22416.527} C_VEL
LIN {X 0,Y 180.395,Z 622.275,A -85,B 0,C 180,E1 -22419.557,E2 -22419.557} C_VEL
LIN {X 0,Y 178.591,Z 620.352,A -85,B 0,C 180,E1 -22422.611,E2 -22422.611} C_VEL
LIN {X 0,Y 178.831,Z 618.674,A -85,B 0,C 180,E1 -22424.428,E2 -22424.428} C_VEL
LIN {X 0,Y 180.69,Z 615.309,A -85,B 0,C 180,E1 -22427.253,E2 -22427.253} C_VEL
LIN {X 0,Y 183.171,Z 615.354,A -85,B 0,C 180,E1 -22430.202,E2 -22430.202} C_VEL
LIN {X 0,Y 188.097,Z 614.162,A -85,B 0,C 180,E1 -22434.269,E2 -22434.269} C_VEL
LIN {X 0,Y 190.955,Z 613.02,A -85,B 0,C 180,E1 -22436.211,E2 -22436.211} C_VEL
LIN {X 0,Y 194.162,Z 611.438,A -85,B 0,C 180,E1 -22438.071,E2 -22438.071} C_VEL
LIN {X 0,Y 199.599,Z 608.371,A -85,B 0,C 180,E1 -22440.702,E2 -22440.702} C_VEL
LIN {X 0,Y 201.348,Z 607.235,A -85,B 0,C 180,E1 -22441.573,E2 -22441.573} C_VEL
LIN {X 0,Y 205.353,Z 603.452,A -85,B 0,C 180,E1 -22444.465,E2 -22444.465} C_VEL
LIN {X 0,Y 208.516,Z 599.663,A -85,B 0,C 180,E1 -22447.351,E2 -22447.351} C_VEL
LIN {X 0,Y 210.375,Z 597.216,A -85,B 0,C 180,E1 -22449.401,E2 -22449.401} C_VEL
LIN {X 0,Y 211.23,Z 595.286,A -85,B 0,C 180,E1 -22451.717,E2 -22451.717} C_VEL
LIN {X 0,Y 211.461,Z 594.031,A -85,B 0,C 180,E1 -22454.264,E2 -22454.264} C_VEL
LIN {X 0,Y 211.638,Z 593.272,A -85,B 0,C 180,E1 -22456.935,E2 -22456.935} C_VEL
LIN {X 0,Y 211.759,Z 593.105,A -85,B 0,C 180,E1 -22459.761,E2 -22459.761} C_VEL
LIN {X 0,Y 211.753,Z 593.264,A -85,B 0,C 180,E1 -22460.906,E2 -22460.906} C_VEL
LIN {X 0,Y 211.403,Z 594.009,A -85,B 0,C 180,E1 -22463.245,E2 -22463.245} C_VEL
LIN {X 0,Y 210.505,Z 595.142,A -85,B 0,C 180,E1 -22465.419,E2 -22465.419} C_VEL
LIN {X 0,Y 209.372,Z 596.658,A -85,B 0,C 180,E1 -22467.516,E2 -22467.516} C_VEL
LIN {X 0,Y 206.42,Z 598.61,A -85,B 0,C 180,E1 -22469.289,E2 -22469.289} C_VEL
LIN {X 0,Y 198.767,Z 602.397,A -85,B 0,C 180,E1 -22472.635,E2 -22472.635} C_VEL
LIN {X 0,Y 195.328,Z 603.575,A -85,B 0,C 180,E1 -22474.421,E2 -22474.421} C_VEL
LIN {X 0,Y 189.219,Z 604.771,A -85,B 0,C 180,E1 -22478.197,E2 -22478.197} C_VEL
LIN {X 0,Y 186.625,Z 604.792,A -85,B 0,C 180,E1 -22480.189,E2 -22480.189} C_VEL
LIN {X 0,Y 182.272,Z 603.503,A -85,B 0,C 180,E1 -22484.342,E2 -22484.342} C_VEL
LIN {X 0,Y 180.395,Z 602.317,A -85,B 0,C 180,E1 -22486.482,E2 -22486.482} C_VEL
LIN {X 0,Y 178.718,Z 600.006,A -85,B 0,C 180,E1 -22489.461,E2 -22489.461} C_VEL
LIN {X 0,Y 177.497,Z 596.063,A -85,B 0,C 180,E1 -22493.178,E2 -22493.178} C_VEL
LIN {X 0,Y 176.883,Z 591.324,A -85,B 0,C 180,E1 -22496.583,E2 -22496.583} C_VEL
LIN {X 0,Y 176.722,Z 585.377,A -85,B 0,C 180,E1 -22500,E2 -22500} C_VEL
LIN {X 0,Y 176.922,Z 579.207,A -85,B 0,C 180,E1 -22502.846,E2 -22502.846} C_VEL
LIN {X 0,Y 177.352,Z 570.031,A -85,B 0,C 180,E1 -22506.256,E2 -22506.256} C_VEL
LIN {X 0,Y 177.856,Z 561.779,A -85,B 0,C 180,E1 -22508.718,E2 -22508.718} C_VEL
LIN {X 0,Y 178.405,Z 553.474,A -85,B 0,C 180,E1 -22510.785,E2 -22510.785} C_VEL
LIN {X 0,Y 179.142,Z 543.79,A -85,B 0,C 180,E1 -22512.749,E2 -22512.749} C_VEL
LIN {X 0,Y 178.794,Z 539.241,A -85,B 0,C 180,E1 -22513.497,E2 -22513.497} C_VEL
LIN {X 0,Y 178.326,Z 536.587,A -85,B 0,C 180,E1 -22513.896,E2 -22513.896} C_VEL
LIN {X 0,Y 178.754,Z 539.082,A -85,B 0,C 180,E1 -22514.37,E2 -22514.37} C_VEL
LIN {X 0,Y 179.389,Z 540.074,A -85,B 0,C 180,E1 -22514.753,E2 -22514.753} C_VEL
LIN {X 0,Y 182.626,Z 540.221,A -85,B 0,C 180,E1 -22516.041,E2 -22516.041} C_VEL
LIN {X 0,Y 185.376,Z 544.389,A -85,B 0,C 180,E1 -22517.656,E2 -22517.656} C_VEL
LIN {X 0,Y 189.878,Z 552.803,A -85,B 0,C 180,E1 -22520.481,E2 -22520.481} C_VEL
LIN {X 0,Y 191.972,Z 557.901,A -85,B 0,C 180,E1 -22522.04,E2 -22522.04} C_VEL
LIN {X 0,Y 193.042,Z 566.122,A -85,B 0,C 180,E1 -22524.122,E2 -22524.122} C_VEL
LIN {X 0,Y 193.271,Z 573.827,A -85,B 0,C 180,E1 -22526.162,E2 -22526.162} C_VEL
LIN {X 0,Y 192.865,Z 580.197,A -85,B 0,C 180,E1 -22527.98,E2 -22527.98} C_VEL
LIN {X 0,Y 192.003,Z 584.082,A -85,B 0,C 180,E1 -22529.082,E2 -22529.082} C_VEL
LIN {X 0,Y 188.962,Z 591.541,A -85,B 0,C 180,E1 -22531.379,E2 -22531.379} C_VEL
LIN {X 0,Y 186.109,Z 597.706,A -85,B 0,C 180,E1 -22533.819,E2 -22533.819} C_VEL
LIN {X 0,Y 183.529,Z 602.92,A -85,B 0,C 180,E1 -22536.468,E2 -22536.468} C_VEL
LIN {X 0,Y 181.327,Z 607.019,A -85,B 0,C 180,E1 -22539.177,E2 -22539.177} C_VEL
LIN {X 0,Y 179.541,Z 610.134,A -85,B 0,C 180,E1 -22541.947,E2 -22541.947} C_VEL
LIN {X 0,Y 177.85,Z 612.757,A -85,B 0,C 180,E1 -22545.341,E2 -22545.341} C_VEL
LIN {X 0,Y 176.584,Z 614.193,A -85,B 0,C 180,E1 -22549.13,E2 -22549.13} C_VEL
LIN {X 0,Y 175.805,Z 614.198,A -85,B 0,C 180,E1 -22553.154,E2 -22553.154} C_VEL
LIN {X 0,Y 175.625,Z 612.764,A -85,B 0,C 180,E1 -22557.178,E2 -22557.178} C_VEL
LIN {X 0,Y 175.915,Z 610.724,A -85,B 0,C 180,E1 -22560.041,E2 -22560.041} C_VEL
LIN {X 0,Y 176.432,Z 607.997,A -85,B 0,C 180,E1 -22562.735,E2 -22562.735} C_VEL
LIN {X 0,Y 177.17,Z 603.735,A -85,B 0,C 180,E1 -22565.835,E2 -22565.835} C_VEL
LIN {X 0,Y 178.112,Z 598.817,A -85,B 0,C 180,E1 -22568.592,E2 -22568.592} C_VEL
LIN {X 0,Y 179.217,Z 593.11,A -85,B 0,C 180,E1 -22571.15,E2 -22571.15} C_VEL
LIN {X 0,Y 180.297,Z 588.127,A -85,B 0,C 180,E1 -22573,E2 -22573} C_VEL
LIN {X 0,Y 181.719,Z 580.891,A -85,B 0,C 180,E1 -22575.213,E2 -22575.213} C_VEL
LIN {X 0,Y 183.128,Z 573.827,A -85,B 0,C 180,E1 -22576.968,E2 -22576.968} C_VEL
LIN {X 0,Y 183.523,Z 570.007,A -85,B 0,C 180,E1 -22577.84,E2 -22577.84} C_VEL
LIN {X 0,Y 182.769,Z 560.46,A -85,B 0,C 180,E1 -22579.755,E2 -22579.755} C_VEL
LIN {X 0,Y 181.884,Z 552.354,A -85,B 0,C 180,E1 -22581.108,E2 -22581.108} C_VEL
LIN {X 0,Y 180.476,Z 543.138,A -85,B 0,C 180,E1 -22582.376,E2 -22582.376} C_VEL
LIN {X 0,Y 178.568,Z 533.547,A -85,B 0,C 180,E1 -22583.431,E2 -22583.431} C_VEL
LIN {X 0,Y 178.414,Z 532.177,A -85,B 0,C 180,E1 -22583.638,E2 -22583.638} C_VEL
LIN {X 0,Y 179.097,Z 526.005,A -85,B 0,C 180,E1 -22588.875,E2 -22588.875} C_VEL
LIN {X 0,Y 179.218,Z 522.973,A -85,B 0,C 180,E1 -22591.544,E2 -22591.544} C_VEL
LIN {X 0,Y 178.936,Z 523.009,A -85,B 0,C 180,E1 -22596.766,E2 -22596.766} C_VEL
LIN {X 0,Y 178.896,Z 523.013,A -85,B 0,C 180,E1 -22600.846,E2 -22600.846} C_VEL
LIN {X 0,Y 178.666,Z 523.042,A -85,B 0,C 180,E1 -22605.982,E2 -22605.982} C_VEL
LIN {X 0,Y 178.624,Z 523.043,A -85,B 0,C 180,E1 -22609.215,E2 -22609.215} C_VEL
LIN {X 0,Y 178.534,Z 523.056,A -85,B 0,C 180,E1 -22615.123,E2 -22615.123} C_VEL
LIN {X 0,Y 178.523,Z 523.06,A -85,B 0,C 180,E1 -22619.993,E2 -22619.993} C_VEL
LIN {X 0,Y 178.496,Z 523.06,A -85,B 0,C 180,E1 -22624.224,E2 -22624.224} C_VEL
LIN {X 0,Y 178.442,Z 523.068,A -85,B 0,C 180,E1 -22629.061,E2 -22629.061} C_VEL
LIN {X 0,Y 178.486,Z 523.059,A -85,B 0,C 180,E1 -22632.018,E2 -22632.018} C_VEL
LIN {X 0,Y 178.515,Z 523.057,A -85,B 0,C 180,E1 -22635.123,E2 -22635.123} C_VEL
LIN {X 0,Y 178.501,Z 523.062,A -85,B 0,C 180,E1 -22638.422,E2 -22638.422} C_VEL
LIN {X 0,Y 178.457,Z 523.059,A -85,B 0,C 180,E1 -22643.791,E2 -22643.791} C_VEL
LIN {X 0,Y 178.488,Z 523.062,A -85,B 0,C 180,E1 -22646.547,E2 -22646.547} C_VEL
LIN {X 0,Y 178.519,Z 523.061,A -85,B 0,C 180,E1 -22650.006,E2 -22650.006} C_VEL
LIN {X 0,Y 178.532,Z 523.056,A -85,B 0,C 180,E1 -22654.875,E2 -22654.875} C_VEL
LIN {X 0,Y 178.621,Z 523.042,A -85,B 0,C 180,E1 -22660.783,E2 -22660.783} C_VEL
LIN {X 0,Y 178.663,Z 523.044,A -85,B 0,C 180,E1 -22664.017,E2 -22664.017} C_VEL
LIN {X 0,Y 178.892,Z 523.008,A -85,B 0,C 180,E1 -22669.153,E2 -22669.153} C_VEL
LIN {X 0,Y 178.932,Z 523.008,A -85,B 0,C 180,E1 -22673.233,E2 -22673.233} C_VEL
LIN {X 0,Y 179.153,Z 522.973,A -85,B 0,C 180,E1 -22677.752,E2 -22677.752} C_VEL
LIN {X 0,Y 179.368,Z 522.948,A -85,B 0,C 180,E1 -22680,E2 -22680} C_VEL
LIN {X 0,Y 178.876,Z 523.015,A -85,B 0,C 180,E1 -22684.507,E2 -22684.507} C_VEL
LIN {X 0,Y 178.976,Z 523.002,A -85,B 0,C 180,E1 -22689.037,E2 -22689.037} C_VEL
LIN {X 0,Y 178.685,Z 523.041,A -85,B 0,C 180,E1 -22693.65,E2 -22693.65} C_VEL
LIN {X 0,Y 178.647,Z 523.045,A -85,B 0,C 180,E1 -22698.344,E2 -22698.344} C_VEL
LIN {X 0,Y 178.509,Z 523.064,A -85,B 0,C 180,E1 -22703.185,E2 -22703.185} C_VEL
LIN {X 0,Y 178.485,Z 523.065,A -85,B 0,C 180,E1 -22708.197,E2 -22708.197} C_VEL
LIN {X 0,Y 178.477,Z 523.066,A -85,B 0,C 180,E1 -22710.791,E2 -22710.791} C_VEL
LIN {X 0,Y 178.494,Z 523.063,A -85,B 0,C 180,E1 -22714.225,E2 -22714.225} C_VEL
LIN {X 0,Y 178.423,Z 523.072,A -85,B 0,C 180,E1 -22719.067,E2 -22719.067} C_VEL
LIN {X 0,Y 178.429,Z 523.073,A -85,B 0,C 180,E1 -22722.036,E2 -22722.036} C_VEL
LIN {X 0,Y 178.459,Z 523.068,A -85,B 0,C 180,E1 -22725.143,E2 -22725.143} C_VEL
LIN {X 0,Y 178.694,Z 523.04,A -85,B 0,C 180,E1 -22731.005,E2 -22731.005} C_VEL
LIN {X 0,Y 179.251,Z 522.973,A -85,B 0,C 180,E1 -22736.315,E2 -22736.315} C_VEL
LIN {X 0,Y 179.253,Z 524.206,A -85,B 0,C 180,E1 -22737.546,E2 -22737.546} C_VEL
LIN {X 0,Y 179.183,Z 530.052,A -85,B 0,C 180,E1 -22739.949,E2 -22739.949} C_VEL
LIN {X 0,Y 178.922,Z 536.74,A -85,B 0,C 180,E1 -22742.517,E2 -22742.517} C_VEL
LIN {X 0,Y 180.927,Z 549.822,A -85,B 0,C 180,E1 -22743.648,E2 -22743.648} C_VEL
LIN {X 0,Y 181.651,Z 559.764,A -85,B 0,C 180,E1 -22744.814,E2 -22744.814} C_VEL
LIN {X 0,Y 181.971,Z 568.287,A -85,B 0,C 180,E1 -22746.077,E2 -22746.077} C_VEL
LIN {X 0,Y 182.024,Z 576.638,A -85,B 0,C 180,E1 -22747.595,E2 -22747.595} C_VEL
LIN {X 0,Y 181.885,Z 583.998,A -85,B 0,C 180,E1 -22749.21,E2 -22749.21} C_VEL
LIN {X 0,Y 181.575,Z 588.051,A -85,B 0,C 180,E1 -22750.205,E2 -22750.205} C_VEL
LIN {X 0,Y 180.016,Z 595.654,A -85,B 0,C 180,E1 -22752.389,E2 -22752.389} C_VEL
LIN {X 0,Y 178.754,Z 601.914,A -85,B 0,C 180,E1 -22754.611,E2 -22754.611} C_VEL
LIN {X 0,Y 177.792,Z 607.112,A -85,B 0,C 180,E1 -22756.863,E2 -22756.863} C_VEL
LIN {X 0,Y 176.891,Z 612.377,A -85,B 0,C 180,E1 -22759.702,E2 -22759.702} C_VEL
LIN {X 0,Y 176.407,Z 615.74,A -85,B 0,C 180,E1 -22761.986,E2 -22761.986} C_VEL
LIN {X 0,Y 176.155,Z 618.456,A -85,B 0,C 180,E1 -22764.277,E2 -22764.277} C_VEL
LIN {X 0,Y 176.064,Z 620.401,A -85,B 0,C 180,E1 -22766.31,E2 -22766.31} C_VEL
LIN {X 0,Y 176.169,Z 622.637,A -85,B 0,C 180,E1 -22770.001,E2 -22770.001} C_VEL
LIN {X 0,Y 176.033,Z 623.535,A -85,B 0,C 180,E1 -22773.53,E2 -22773.53} C_VEL
LIN {X 0,Y 176.323,Z 623.31,A -85,B 0,C 180,E1 -22776.869,E2 -22776.869} C_VEL
LIN {X 0,Y 176.737,Z 622.502,A -85,B 0,C 180,E1 -22779.154,E2 -22779.154} C_VEL
LIN {X 0,Y 177.445,Z 621.225,A -85,B 0,C 180,E1 -22781.423,E2 -22781.423} C_VEL
LIN {X 0,Y 178.831,Z 618.674,A -85,B 0,C 180,E1 -22784.428,E2 -22784.428} C_VEL
LIN {X 0,Y 178.866,Z 617.49,A -85,B 0,C 180,E1 -22785.658,E2 -22785.658} C_VEL
LIN {X 0,Y 177.333,Z 615.944,A -85,B 0,C 180,E1 -22787.733,E2 -22787.733} C_VEL
LIN {X 0,Y 176.145,Z 615.012,A -85,B 0,C 180,E1 -22789.867,E2 -22789.867} C_VEL
LIN {X 0,Y 176.698,Z 614.794,A -85,B 0,C 180,E1 -22791.144,E2 -22791.144} C_VEL
LIN {X 0,Y 178.948,Z 614.701,A -85,B 0,C 180,E1 -22793.126,E2 -22793.126} C_VEL
LIN {X 0,Y 184.618,Z 613.204,A -85,B 0,C 180,E1 -22797.183,E2 -22797.183} C_VEL
LIN {X 0,Y 187.959,Z 611.987,A -85,B 0,C 180,E1 -22799.085,E2 -22799.085} C_VEL
LIN {X 0,Y 193.591,Z 609.343,A -85,B 0,C 180,E1 -22801.764,E2 -22801.764} C_VEL
LIN {X 0,Y 195.376,Z 608.255,A -85,B 0,C 180,E1 -22802.656,E2 -22802.656} C_VEL
LIN {X 0,Y 198.184,Z 606.176,A -85,B 0,C 180,E1 -22804.57,E2 -22804.57} C_VEL
LIN {X 0,Y 201.809,Z 602.781,A -85,B 0,C 180,E1 -22807.55,E2 -22807.55} C_VEL
LIN {X 0,Y 203.932,Z 600.515,A -85,B 0,C 180,E1 -22809.611,E2 -22809.611} C_VEL
LIN {X 0,Y 204.64,Z 599.44,A -85,B 0,C 180,E1 -22810.927,E2 -22810.927} C_VEL
LIN {X 0,Y 205.267,Z 598.07,A -85,B 0,C 180,E1 -22813.219,E2 -22813.219} C_VEL
LIN {X 0,Y 205.539,Z 596.948,A -85,B 0,C 180,E1 -22816.854,E2 -22816.854} C_VEL
LIN {X 0,Y 205.622,Z 596.672,A -85,B 0,C 180,E1 -22819.504,E2 -22819.504} C_VEL
LIN {X 0,Y 205.349,Z 597.021,A -85,B 0,C 180,E1 -22821.972,E2 -22821.972} C_VEL
LIN {X 0,Y 204.58,Z 597.897,A -85,B 0,C 180,E1 -22824.267,E2 -22824.267} C_VEL
LIN {X 0,Y 203.38,Z 598.896,A -85,B 0,C 180,E1 -22826.434,E2 -22826.434} C_VEL
LIN {X 0,Y 200.541,Z 600.638,A -85,B 0,C 180,E1 -22828.286,E2 -22828.286} C_VEL
LIN {X 0,Y 196.452,Z 602.386,A -85,B 0,C 180,E1 -22829.944,E2 -22829.944} C_VEL
LIN {X 0,Y 189.025,Z 604.665,A -85,B 0,C 180,E1 -22833.502,E2 -22833.502} C_VEL
LIN {X 0,Y 185.709,Z 605.251,A -85,B 0,C 180,E1 -22835.4,E2 -22835.4} C_VEL
LIN {X 0,Y 179.97,Z 605.077,A -85,B 0,C 180,E1 -22839.424,E2 -22839.424} C_VEL
LIN {X 0,Y 177.562,Z 604.478,A -85,B 0,C 180,E1 -22841.54,E2 -22841.54} C_VEL
LIN {X 0,Y 173.534,Z 601.893,A -85,B 0,C 180,E1 -22845.937,E2 -22845.937} C_VEL
LIN {X 0,Y 171.674,Z 599.027,A -85,B 0,C 180,E1 -22849.275,E2 -22849.275} C_VEL
LIN {X 0,Y 170.531,Z 595.013,A -85,B 0,C 180,E1 -22852.898,E2 -22852.898} C_VEL
LIN {X 0,Y 170.118,Z 591.795,A -85,B 0,C 180,E1 -22855.261,E2 -22855.261} C_VEL
LIN {X 0,Y 169.761,Z 585.853,A -85,B 0,C 180,E1 -22858.814,E2 -22858.814} C_VEL
LIN {X 0,Y 169.942,Z 578.552,A -85,B 0,C 180,E1 -22862.37,E2 -22862.37} C_VEL
LIN {X 0,Y 170.253,Z 570.885,A -85,B 0,C 180,E1 -22865.329,E2 -22865.329} C_VEL
LIN {X 0,Y 170.8,Z 562.355,A -85,B 0,C 180,E1 -22868.004,E2 -22868.004} C_VEL
LIN {X 0,Y 171.369,Z 554.056,A -85,B 0,C 180,E1 -22870.172,E2 -22870.172} C_VEL
LIN {X 0,Y 171.991,Z 544.859,A -85,B 0,C 180,E1 -22872.164,E2 -22872.164} C_VEL
LIN {X 0,Y 172.023,Z 547.315,A -85,B 0,C 180,E1 -22872.686,E2 -22872.686} C_VEL
LIN {X 0,Y 173.532,Z 548.458,A -85,B 0,C 180,E1 -22873.587,E2 -22873.587} C_VEL
LIN {X 0,Y 177.252,Z 546.821,A -85,B 0,C 180,E1 -22874.935,E2 -22874.935} C_VEL
LIN {X 0,Y 179.438,Z 547.004,A -85,B 0,C 180,E1 -22875.84,E2 -22875.84} C_VEL
LIN {X 0,Y 181.238,Z 549.923,A -85,B 0,C 180,E1 -22877.031,E2 -22877.031} C_VEL
LIN {X 0,Y 185.166,Z 557.905,A -85,B 0,C 180,E1 -22879.974,E2 -22879.974} C_VEL
LIN {X 0,Y 186.588,Z 561.782,A -85,B 0,C 180,E1 -22881.28,E2 -22881.28} C_VEL
LIN {X 0,Y 187.326,Z 571.468,A -85,B 0,C 180,E1 -22883.932,E2 -22883.932} C_VEL
LIN {X 0,Y 186.99,Z 579.255,A -85,B 0,C 180,E1 -22886.239,E2 -22886.239} C_VEL
LIN {X 0,Y 185.994,Z 584.831,A -85,B 0,C 180,E1 -22887.961,E2 -22887.961} C_VEL
LIN {X 0,Y 182.75,Z 592.229,A -85,B 0,C 180,E1 -22890.343,E2 -22890.343} C_VEL
LIN {X 0,Y 180.175,Z 597.533,A -85,B 0,C 180,E1 -22892.484,E2 -22892.484} C_VEL
LIN {X 0,Y 177.71,Z 602.225,A -85,B 0,C 180,E1 -22894.853,E2 -22894.853} C_VEL
LIN {X 0,Y 175.857,Z 605.586,A -85,B 0,C 180,E1 -22896.936,E2 -22896.936} C_VEL
LIN {X 0,Y 173.211,Z 609.782,A -85,B 0,C 180,E1 -22900.481,E2 -22900.481} C_VEL
LIN {X 0,Y 171.18,Z 612.743,A -85,B 0,C 180,E1 -22904.264,E2 -22904.264} C_VEL
LIN {X 0,Y 169.633,Z 614.388,A -85,B 0,C 180,E1 -22908.478,E2 -22908.478} C_VEL
LIN {X 0,Y 168.809,Z 614.461,A -85,B 0,C 180,E1 -22912.282,E2 -22912.282} C_VEL
LIN {X 0,Y 168.599,Z 614.063,A -85,B 0,C 180,E1 -22914.296,E2 -22914.296} C_VEL
LIN {X 0,Y 168.526,Z 612.805,A -85,B 0,C 180,E1 -22917.169,E2 -22917.169} C_VEL
LIN {X 0,Y 168.936,Z 609.978,A -85,B 0,C 180,E1 -22920.884,E2 -22920.884} C_VEL
LIN {X 0,Y 169.335,Z 608.036,A -85,B 0,C 180,E1 -22922.835,E2 -22922.835} C_VEL
LIN {X 0,Y 170.153,Z 603.419,A -85,B 0,C 180,E1 -22926.251,E2 -22926.251} C_VEL
LIN {X 0,Y 171.282,Z 597.814,A -85,B 0,C 180,E1 -22929.411,E2 -22929.411} C_VEL
LIN {X 0,Y 172.628,Z 591.488,A -85,B 0,C 180,E1 -22932.22,E2 -22932.22} C_VEL
LIN {X 0,Y 174.45,Z 582.779,A -85,B 0,C 180,E1 -22935.213,E2 -22935.213} C_VEL
LIN {X 0,Y 176.091,Z 574.868,A -85,B 0,C 180,E1 -22937.319,E2 -22937.319} C_VEL
LIN {X 0,Y 176.611,Z 571.042,A -85,B 0,C 180,E1 -22938.231,E2 -22938.231} C_VEL
LIN {X 0,Y 175.936,Z 561.717,A -85,B 0,C 180,E1 -22940.224,E2 -22940.224} C_VEL
LIN {X 0,Y 175.146,Z 553.759,A -85,B 0,C 180,E1 -22941.635,E2 -22941.635} C_VEL
LIN {X 0,Y 173.569,Z 543.143,A -85,B 0,C 180,E1 -22943.168,E2 -22943.168} C_VEL
LIN {X 0,Y 171.651,Z 533.594,A -85,B 0,C 180,E1 -22944.271,E2 -22944.271} C_VEL
LIN {X 0,Y 171.46,Z 532.398,A -85,B 0,C 180,E1 -22944.412,E2 -22944.412} C_VEL
LIN {X 0,Y 172.25,Z 526.027,A -85,B 0,C 180,E1 -22949.999,E2 -22949.999} C_VEL
LIN {X 0,Y 172.148,Z 523.854,A -85,B 0,C 180,E1 -22952.046,E2 -22952.046} C_VEL
LIN {X 0,Y 171.901,Z 523.885,A -85,B 0,C 180,E1 -22957.044,E2 -22957.044} C_VEL
LIN {X 0,Y 171.851,Z 523.89,A -85,B 0,C 180,E1 -22961.037,E2 -22961.037} C_VEL
LIN {X 0,Y 171.586,Z 523.923,A -85,B 0,C 180,E1 -22966.66,E2 -22966.66} C_VEL
LIN {X 0,Y 171.545,Z 523.925,A -85,B 0,C 180,E1 -22969.561,E2 -22969.561} C_VEL
LIN {X 0,Y 171.469,Z 523.937,A -85,B 0,C 180,E1 -22975.615,E2 -22975.615} C_VEL
LIN {X 0,Y 171.441,Z 523.942,A -85,B 0,C 180,E1 -22980.586,E2 -22980.586} C_VEL
LIN {X 0,Y 171.406,Z 523.941,A -85,B 0,C 180,E1 -22985.03,E2 -22985.03} C_VEL
LIN {X 0,Y 171.399,Z 523.946,A -85,B 0,C 180,E1 -22988.824,E2 -22988.824} C_VEL
LIN {X 0,Y 171.438,Z 523.938,A -85,B 0,C 180,E1 -22994.178,E2 -22994.178} C_VEL
LIN {X 0,Y 171.418,Z 523.943,A -85,B 0,C 180,E1 -22999.005,E2 -22999.005} C_VEL
LIN {X 0,Y 171.435,Z 523.935,A -85,B 0,C 180,E1 -23002.053,E2 -23002.053} C_VEL
LIN {X 0,Y 171.416,Z 523.945,A -85,B 0,C 180,E1 -23007.792,E2 -23007.792} C_VEL
LIN {X 0,Y 171.445,Z 523.94,A -85,B 0,C 180,E1 -23010.533,E2 -23010.533} C_VEL
LIN {X 0,Y 171.455,Z 523.94,A -85,B 0,C 180,E1 -23015.801,E2 -23015.801} C_VEL
LIN {X 0,Y 171.577,Z 523.919,A -85,B 0,C 180,E1 -23020.871,E2 -23020.871} C_VEL
LIN {X 0,Y 171.608,Z 523.923,A -85,B 0,C 180,E1 -23025.775,E2 -23025.775} C_VEL
LIN {X 0,Y 171.908,Z 523.882,A -85,B 0,C 180,E1 -23030.588,E2 -23030.588} C_VEL
LIN {X 0,Y 171.825,Z 523.893,A -85,B 0,C 180,E1 -23035.308,E2 -23035.308} C_VEL
LIN {X 0,Y 172.331,Z 523.824,A -85,B 0,C 180,E1 -23040,E2 -23040} C_VEL
LIN {X 0,Y 171.825,Z 523.893,A -85,B 0,C 180,E1 -23044.692,E2 -23044.692} C_VEL
LIN {X 0,Y 171.908,Z 523.884,A -85,B 0,C 180,E1 -23049.412,E2 -23049.412} C_VEL
LIN {X 0,Y 171.607,Z 523.922,A -85,B 0,C 180,E1 -23054.224,E2 -23054.224} C_VEL
LIN {X 0,Y 171.542,Z 523.933,A -85,B 0,C 180,E1 -23059.563,E2 -23059.563} C_VEL
LIN {X 0,Y 171.467,Z 523.942,A -85,B 0,C 180,E1 -23065.617,E2 -23065.617} C_VEL
LIN {X 0,Y 171.439,Z 523.943,A -85,B 0,C 180,E1 -23070.587,E2 -23070.587} C_VEL
LIN {X 0,Y 171.404,Z 523.946,A -85,B 0,C 180,E1 -23075.032,E2 -23075.032} C_VEL
LIN {X 0,Y 171.383,Z 523.948,A -85,B 0,C 180,E1 -23078.82,E2 -23078.82} C_VEL
LIN {X 0,Y 171.368,Z 523.951,A -85,B 0,C 180,E1 -23084.202,E2 -23084.202} C_VEL
LIN {X 0,Y 171.516,Z 523.933,A -85,B 0,C 180,E1 -23089.036,E2 -23089.036} C_VEL
LIN {X 0,Y 172.127,Z 523.86,A -85,B 0,C 180,E1 -23095.138,E2 -23095.138} C_VEL
LIN {X 0,Y 172.233,Z 523.903,A -85,B 0,C 180,E1 -23096.224,E2 -23096.224} C_VEL
LIN {X 0,Y 172.531,Z 527.811,A -85,B 0,C 180,E1 -23098.026,E2 -23098.026} C_VEL
LIN {X 0,Y 172.069,Z 536.421,A -85,B 0,C 180,E1 -23101.637,E2 -23101.637} C_VEL
LIN {X 0,Y 174.073,Z 550.138,A -85,B 0,C 180,E1 -23102.927,E2 -23102.927} C_VEL
LIN {X 0,Y 174.773,Z 559.443,A -85,B 0,C 180,E1 -23104.069,E2 -23104.069} C_VEL
LIN {X 0,Y 175.072,Z 568.031,A -85,B 0,C 180,E1 -23105.388,E2 -23105.388} C_VEL
LIN {X 0,Y 175.102,Z 577.154,A -85,B 0,C 180,E1 -23107.121,E2 -23107.121} C_VEL
LIN {X 0,Y 174.859,Z 585.654,A -85,B 0,C 180,E1 -23109.103,E2 -23109.103} C_VEL
LIN {X 0,Y 173.641,Z 592.878,A -85,B 0,C 180,E1 -23111.109,E2 -23111.109} C_VEL
LIN {X 0,Y 171.872,Z 601.019,A -85,B 0,C 180,E1 -23113.979,E2 -23113.979} C_VEL
LIN {X 0,Y 170.857,Z 606.334,A -85,B 0,C 180,E1 -23116.32,E2 -23116.32} C_VEL
LIN {X 0,Y 169.897,Z 611.703,A -85,B 0,C 180,E1 -23119.273,E2 -23119.273} C_VEL
LIN {X 0,Y 169.377,Z 615.163,A -85,B 0,C 180,E1 -23121.651,E2 -23121.651} C_VEL
LIN {X 0,Y 169.005,Z 619.105,A -85,B 0,C 180,E1 -23125.23,E2 -23125.23} C_VEL
LIN {X 0,Y 168.975,Z 620.974,A -85,B 0,C 180,E1 -23127.617,E2 -23127.617} C_VEL
LIN {X 0,Y 169.074,Z 622.318,A -85,B 0,C 180,E1 -23130.001,E2 -23130.001} C_VEL
LIN {X 0,Y 168.931,Z 623.243,A -85,B 0,C 180,E1 -23133.179,E2 -23133.179} C_VEL
LIN {X 0,Y 169.007,Z 623.422,A -85,B 0,C 180,E1 -23134.772,E2 -23134.772} C_VEL
LIN {X 0,Y 169.267,Z 623.158,A -85,B 0,C 180,E1 -23137.157,E2 -23137.157} C_VEL
LIN {X 0,Y 169.718,Z 622.434,A -85,B 0,C 180,E1 -23139.536,E2 -23139.536} C_VEL
LIN {X 0,Y 170.471,Z 621.243,A -85,B 0,C 180,E1 -23141.897,E2 -23141.897} C_VEL
LIN {X 0,Y 172.176,Z 618.417,A -85,B 0,C 180,E1 -23145.387,E2 -23145.387} C_VEL
LIN {X 0,Y 174.51,Z 614.612,A -85,B 0,C 180,E1 -23148.644,E2 -23148.644} C_VEL
LIN {X 0,Y 176.698,Z 614.794,A -85,B 0,C 180,E1 -23151.144,E2 -23151.144} C_VEL
LIN {X 0,Y 178.082,Z 614.712,A -85,B 0,C 180,E1 -23153.001,E2 -23153.001} C_VEL
LIN {X 0,Y 180.313,Z 613.048,A -85,B 0,C 180,E1 -23158.639,E2 -23158.639} C_VEL
LIN {X 0,Y 182.289,Z 612.145,A -85,B 0,C 180,E1 -23160.362,E2 -23160.362} C_VEL
LIN {X 0,Y 183.249,Z 611.746,A -85,B 0,C 180,E1 -23160.885,E2 -23160.885} C_VEL
LIN {X 0,Y 189.455,Z 609.227,A -85,B 0,C 180,E1 -23163.811,E2 -23163.811} C_VEL
LIN {X 0,Y 192.35,Z 607.307,A -85,B 0,C 180,E1 -23165.776,E2 -23165.776} C_VEL
LIN {X 0,Y 194.971,Z 605.419,A -85,B 0,C 180,E1 -23167.793,E2 -23167.793} C_VEL
LIN {X 0,Y 197.288,Z 603.385,A -85,B 0,C 180,E1 -23169.884,E2 -23169.884} C_VEL
LIN {X 0,Y 198.528,Z 601.797,A -85,B 0,C 180,E1 -23172.27,E2 -23172.27} C_VEL
LIN {X 0,Y 199.091,Z 600.67,A -85,B 0,C 180,E1 -23175.089,E2 -23175.089} C_VEL
LIN {X 0,Y 199.259,Z 600.067,A -85,B 0,C 180,E1 -23177.922,E2 -23177.922} C_VEL
LIN {X 0,Y 199.062,Z 599.995,A -85,B 0,C 180,E1 -23180.963,E2 -23180.963} C_VEL
LIN {X 0,Y 198.448,Z 600.365,A -85,B 0,C 180,E1 -23182.983,E2 -23182.983} C_VEL
LIN {X 0,Y 197.382,Z 601.191,A -85,B 0,C 180,E1 -23185.271,E2 -23185.271} C_VEL
LIN {X 0,Y 194.686,Z 602.363,A -85,B 0,C 180,E1 -23187.215,E2 -23187.215} C_VEL
LIN {X 0,Y 186.477,Z 604.996,A -85,B 0,C 180,E1 -23190.663,E2 -23190.663} C_VEL
LIN {X 0,Y 179.299,Z 605.873,A -85,B 0,C 180,E1 -23194.458,E2 -23194.458} C_VEL
LIN {X 0,Y 176.182,Z 605.821,A -85,B 0,C 180,E1 -23196.49,E2 -23196.49} C_VEL
LIN {X 0,Y 170.852,Z 604.349,A -85,B 0,C 180,E1 -23200.787,E2 -23200.787} C_VEL
LIN {X 0,Y 168.671,Z 603.108,A -85,B 0,C 180,E1 -23203.042,E2 -23203.042} C_VEL
LIN {X 0,Y 165.945,Z 600.404,A -85,B 0,C 180,E1 -23206.53,E2 -23206.53} C_VEL
LIN {X 0,Y 164.248,Z 596.778,A -85,B 0,C 180,E1 -23210.145,E2 -23210.145} C_VEL
LIN {X 0,Y 163.363,Z 592.133,A -85,B 0,C 180,E1 -23213.826,E2 -23213.826} C_VEL
LIN {X 0,Y 162.865,Z 586.315,A -85,B 0,C 180,E1 -23217.527,E2 -23217.527} C_VEL
LIN {X 0,Y 162.981,Z 579.054,A -85,B 0,C 180,E1 -23221.236,E2 -23221.236} C_VEL
LIN {X 0,Y 163.332,Z 569.797,A -85,B 0,C 180,E1 -23224.937,E2 -23224.937} C_VEL
LIN {X 0,Y 163.853,Z 561.267,A -85,B 0,C 180,E1 -23227.713,E2 -23227.713} C_VEL
LIN {X 0,Y 164.406,Z 552.737,A -85,B 0,C 180,E1 -23229.975,E2 -23229.975} C_VEL
LIN {X 0,Y 164.275,Z 554.04,A -85,B 0,C 180,E1 -23230.261,E2 -23230.261} C_VEL
LIN {X 0,Y 164.494,Z 555.131,A -85,B 0,C 180,E1 -23230.675,E2 -23230.675} C_VEL
LIN {X 0,Y 167.08,Z 555.514,A -85,B 0,C 180,E1 -23232.141,E2 -23232.141} C_VEL
LIN {X 0,Y 169.746,Z 554.372,A -85,B 0,C 180,E1 -23233.163,E2 -23233.163} C_VEL
LIN {X 0,Y 171.695,Z 555.047,A -85,B 0,C 180,E1 -23234.217,E2 -23234.217} C_VEL
LIN {X 0,Y 174.949,Z 553.936,A -85,B 0,C 180,E1 -23235.391,E2 -23235.391} C_VEL
LIN {X 0,Y 176.563,Z 554.577,A -85,B 0,C 180,E1 -23236.179,E2 -23236.179} C_VEL
LIN {X 0,Y 179.607,Z 561.093,A -85,B 0,C 180,E1 -23238.834,E2 -23238.834} C_VEL
LIN {X 0,Y 181.123,Z 565.436,A -85,B 0,C 180,E1 -23240.44,E2 -23240.44} C_VEL
LIN {X 0,Y 181.436,Z 573.293,A -85,B 0,C 180,E1 -23242.79,E2 -23242.79} C_VEL
LIN {X 0,Y 180.85,Z 581.189,A -85,B 0,C 180,E1 -23245.307,E2 -23245.307} C_VEL
LIN {X 0,Y 180.371,Z 584.295,A -85,B 0,C 180,E1 -23246.338,E2 -23246.338} C_VEL
LIN {X 0,Y 178.292,Z 589.432,A -85,B 0,C 180,E1 -23247.991,E2 -23247.991} C_VEL
LIN {X 0,Y 174.352,Z 597.367,A -85,B 0,C 180,E1 -23251.064,E2 -23251.064} C_VEL
LIN {X 0,Y 171.317,Z 602.701,A -85,B 0,C 180,E1 -23253.837,E2 -23253.837} C_VEL
LIN {X 0,Y 168.978,Z 606.535,A -85,B 0,C 180,E1 -23256.403,E2 -23256.403} C_VEL
LIN {X 0,Y 166.054,Z 610.813,A -85,B 0,C 180,E1 -23260.373,E2 -23260.373} C_VEL
LIN {X 0,Y 164.434,Z 612.94,A -85,B 0,C 180,E1 -23263.397,E2 -23263.397} C_VEL
LIN {X 0,Y 162.894,Z 614.492,A -85,B 0,C 180,E1 -23267.177,E2 -23267.177} C_VEL
LIN {X 0,Y 161.834,Z 614.712,A -85,B 0,C 180,E1 -23271.416,E2 -23271.416} C_VEL
LIN {X 0,Y 161.427,Z 613.497,A -85,B 0,C 180,E1 -23275.812,E2 -23275.812} C_VEL
LIN {X 0,Y 161.75,Z 610.562,A -85,B 0,C 180,E1 -23280.343,E2 -23280.343} C_VEL
LIN {X 0,Y 162.247,Z 608.061,A -85,B 0,C 180,E1 -23282.945,E2 -23282.945} C_VEL
LIN {X 0,Y 163.019,Z 603.931,A -85,B 0,C 180,E1 -23286.155,E2 -23286.155} C_VEL
LIN {X 0,Y 164.077,Z 598.679,A -85,B 0,C 180,E1 -23289.305,E2 -23289.305} C_VEL
LIN {X 0,Y 165.313,Z 592.929,A -85,B 0,C 180,E1 -23292.047,E2 -23292.047} C_VEL
LIN {X 0,Y 166.939,Z 585.939,A -85,B 0,C 180,E1 -23294.719,E2 -23294.719} C_VEL
LIN {X 0,Y 168.79,Z 577.151,A -85,B 0,C 180,E1 -23297.372,E2 -23297.372} C_VEL
LIN {X 0,Y 169.684,Z 571.942,A -85,B 0,C 180,E1 -23298.653,E2 -23298.653} C_VEL
LIN {X 0,Y 168.982,Z 561.342,A -85,B 0,C 180,E1 -23301.026,E2 -23301.026} C_VEL
LIN {X 0,Y 168.142,Z 553.362,A -85,B 0,C 180,E1 -23302.493,E2 -23302.493} C_VEL
LIN {X 0,Y 166.637,Z 543.238,A -85,B 0,C 180,E1 -23304.022,E2 -23304.022} C_VEL
LIN {X 0,Y 164.735,Z 533.725,A -85,B 0,C 180,E1 -23305.181,E2 -23305.181} C_VEL
LIN {X 0,Y 164.555,Z 532.447,A -85,B 0,C 180,E1 -23305.406,E2 -23305.406} C_VEL
LIN {X 0,Y 165.225,Z 527.357,A -85,B 0,C 180,E1 -23309.999,E2 -23309.999} C_VEL
LIN {X 0,Y 165.313,Z 526.049,A -85,B 0,C 180,E1 -23311.217,E2 -23311.217} C_VEL
LIN {X 0,Y 165.006,Z 524.746,A -85,B 0,C 180,E1 -23312.593,E2 -23312.593} C_VEL
LIN {X 0,Y 164.864,Z 524.762,A -85,B 0,C 180,E1 -23317.346,E2 -23317.346} C_VEL
LIN {X 0,Y 164.781,Z 524.771,A -85,B 0,C 180,E1 -23321.197,E2 -23321.197} C_VEL
LIN {X 0,Y 164.506,Z 524.804,A -85,B 0,C 180,E1 -23327.399,E2 -23327.399} C_VEL
LIN {X 0,Y 164.474,Z 524.807,A -85,B 0,C 180,E1 -23329.988,E2 -23329.988} C_VEL
LIN {X 0,Y 164.394,Z 524.82,A -85,B 0,C 180,E1 -23336.133,E2 -23336.133} C_VEL
LIN {X 0,Y 164.376,Z 524.821,A -85,B 0,C 180,E1 -23341.227,E2 -23341.227} C_VEL
LIN {X 0,Y 164.339,Z 524.825,A -85,B 0,C 180,E1 -23346.776,E2 -23346.776} C_VEL
LIN {X 0,Y 164.337,Z 524.827,A -85,B 0,C 180,E1 -23349.901,E2 -23349.901} C_VEL
LIN {X 0,Y 164.371,Z 524.814,A -85,B 0,C 180,E1 -23353.375,E2 -23353.375} C_VEL
LIN {X 0,Y 164.382,Z 524.82,A -85,B 0,C 180,E1 -23356.838,E2 -23356.838} C_VEL
LIN {X 0,Y 164.369,Z 524.819,A -85,B 0,C 180,E1 -23360.319,E2 -23360.319} C_VEL
LIN {X 0,Y 164.343,Z 524.819,A -85,B 0,C 180,E1 -23364.341,E2 -23364.341} C_VEL
LIN {X 0,Y 164.387,Z 524.82,A -85,B 0,C 180,E1 -23369.134,E2 -23369.134} C_VEL
LIN {X 0,Y 164.414,Z 524.815,A -85,B 0,C 180,E1 -23374.693,E2 -23374.693} C_VEL
LIN {X 0,Y 164.482,Z 524.805,A -85,B 0,C 180,E1 -23380.05,E2 -23380.05} C_VEL
LIN {X 0,Y 164.551,Z 524.799,A -85,B 0,C 180,E1 -23385.151,E2 -23385.151} C_VEL
LIN {X 0,Y 164.851,Z 524.762,A -85,B 0,C 180,E1 -23390.181,E2 -23390.181} C_VEL
LIN {X 0,Y 164.775,Z 524.77,A -85,B 0,C 180,E1 -23395.106,E2 -23395.106} C_VEL
LIN {X 0,Y 165.294,Z 524.7,A -85,B 0,C 180,E1 -23400,E2 -23400} C_VEL
LIN {X 0,Y 164.775,Z 524.771,A -85,B 0,C 180,E1 -23404.893,E2 -23404.893} C_VEL
LIN {X 0,Y 164.85,Z 524.764,A -85,B 0,C 180,E1 -23409.818,E2 -23409.818} C_VEL
LIN {X 0,Y 164.551,Z 524.8,A -85,B 0,C 180,E1 -23414.848,E2 -23414.848} C_VEL
LIN {X 0,Y 164.471,Z 524.811,A -85,B 0,C 180,E1 -23419.989,E2 -23419.989} C_VEL
LIN {X 0,Y 164.391,Z 524.822,A -85,B 0,C 180,E1 -23426.134,E2 -23426.134} C_VEL
LIN {X 0,Y 164.373,Z 524.824,A -85,B 0,C 180,E1 -23431.229,E2 -23431.229} C_VEL
LIN {X 0,Y 164.312,Z 524.829,A -85,B 0,C 180,E1 -23436.785,E2 -23436.785} C_VEL
LIN {X 0,Y 164.303,Z 524.832,A -85,B 0,C 180,E1 -23439.912,E2 -23439.912} C_VEL
LIN {X 0,Y 164.304,Z 524.834,A -85,B 0,C 180,E1 -23443.353,E2 -23443.353} C_VEL
LIN {X 0,Y 164.372,Z 524.823,A -85,B 0,C 180,E1 -23446.836,E2 -23446.836} C_VEL
LIN {X 0,Y 164.543,Z 524.802,A -85,B 0,C 180,E1 -23450.248,E2 -23450.248} C_VEL
LIN {X 0,Y 165.132,Z 524.858,A -85,B 0,C 180,E1 -23455.397,E2 -23455.397} C_VEL
LIN {X 0,Y 165.724,Z 529.089,A -85,B 0,C 180,E1 -23457.498,E2 -23457.498} C_VEL
LIN {X 0,Y 165.224,Z 536.582,A -85,B 0,C 180,E1 -23460.787,E2 -23460.787} C_VEL
LIN {X 0,Y 167.14,Z 549.284,A -85,B 0,C 180,E1 -23462.008,E2 -23462.008} C_VEL
LIN {X 0,Y 167.91,Z 558.134,A -85,B 0,C 180,E1 -23463.13,E2 -23463.13} C_VEL
LIN {X 0,Y 168.173,Z 566.45,A -85,B 0,C 180,E1 -23464.419,E2 -23464.419} C_VEL
LIN {X 0,Y 168.233,Z 574.875,A -85,B 0,C 180,E1 -23466.029,E2 -23466.029} C_VEL
LIN {X 0,Y 168.041,Z 582.901,A -85,B 0,C 180,E1 -23467.89,E2 -23467.89} C_VEL
LIN {X 0,Y 167.516,Z 588.62,A -85,B 0,C 180,E1 -23469.43,E2 -23469.43} C_VEL
LIN {X 0,Y 166.097,Z 595.226,A -85,B 0,C 180,E1 -23471.499,E2 -23471.499} C_VEL
LIN {X 0,Y 164.741,Z 601.488,A -85,B 0,C 180,E1 -23473.902,E2 -23473.902} C_VEL
LIN {X 0,Y 163.708,Z 606.689,A -85,B 0,C 180,E1 -23476.344,E2 -23476.344} C_VEL
LIN {X 0,Y 162.919,Z 611.007,A -85,B 0,C 180,E1 -23478.808,E2 -23478.808} C_VEL
LIN {X 0,Y 162.159,Z 616.074,A -85,B 0,C 180,E1 -23482.531,E2 -23482.531} C_VEL
LIN {X 0,Y 161.931,Z 618.609,A -85,B 0,C 180,E1 -23485.022,E2 -23485.022} C_VEL
LIN {X 0,Y 161.884,Z 620.569,A -85,B 0,C 180,E1 -23487.513,E2 -23487.513} C_VEL
LIN {X 0,Y 161.982,Z 621.998,A -85,B 0,C 180,E1 -23490.001,E2 -23490.001} C_VEL
LIN {X 0,Y 161.854,Z 622.965,A -85,B 0,C 180,E1 -23492.924,E2 -23492.924} C_VEL
LIN {X 0,Y 161.934,Z 623.186,A -85,B 0,C 180,E1 -23494.981,E2 -23494.981} C_VEL
